FUNCTION_BLOCK "GCS7_E_MTRI"	// FB 57
TITLE = MTRI
//  
//COPYRIGHT:    (C) 1996 BY  BUHLER LTD.
//                           CH-9240 UZWIL  SWITZERLAND
//
//PRODUCT:      GCS7
//
//TITLE:        Element Control MTRI
//
//-------------------------------------------------------------------------
//
//IDENT:        AUTHOR:             DEPT:                       DATE:
//
//FB57.1.2      A.Egli              CT3                         18-Nov-2003
//              Handling Restdischarge
//FB57.1.1      A.Egli              CT3                         29-Sep-2003
//              Value in Units [1.00 to 8.00] = [-60° to 45°]
//FB57.1.0      A.Egli              CT3                         22-Apr-2003
//              1st Release in S7
//
//-------------------------------------------------------------------------
//
//PURPOSE:      MANUAL : see [MTRIxxMAN]
//
//RESTRICTIONS: S7
//
//-------------------------------------------------------------------------
//
//=======================================================
//Log Message: 
//------------------------------------------------------
//0   Stopped
//2   Adjusted
//9   fault cancelled
//10  emptied
//11  fault monitoring time
//12  fault adjusting time
//13  fault toloerance
//
//=======================================================
//StCode:  State               
//------------------------------------------------------
//32  StFault               
// 1  StStopped             
//41  StStopped.HWStop               StStopped + InHWStop
//51  StStopped.DPFault              StStopped + InDPFault
// 2  StAdjusting             
//12  StAdjusting.Calibration             
// 3  StAdjusted.Automatic              
//13  StAdjusted.Hand
//
AUTHOR : EA
FAMILY : GCS7LL
NAME : MTRI
VERSION : 1.2
VAR
  StCode : INT ;	//Element state code
  InEnable : BOOL ;	//Interlocking: 1=Enable to open /0=Intermediate closing
  CmdRestdischarge : BOOL ;	//Command to restdischarge
  CmdCalibration : BOOL ;	//Calibration 0 point
  InpMinus : BOOL ;	//Input button "Minus"
  InpPlus : BOOL ;	//Input button "Plus"
  CmdNewJob : BOOL ;	//Command new job
  InModeRemote : BOOL ;	//1=Target position from PC, 0=Target position with +/-
  spare27 : BOOL ;
  CmdOff : BOOL ;	//Pulse to stop  (manual mode)
  CmdOn : BOOL ;	//Pulse to start  (manual mode)
  CmdNext : BOOL ;	//Pulse to start element in automatic mode
  CmdFaultReset : BOOL ;	//Command to reset fault
  InLocal : BOOL ;	//1= Local mode (no fault by start with service switch)
  InManual : BOOL ;	//1= Manual/ 0= Automatic
  InReport : BOOL ;	//Report of all state transitions
  spare0207 : BOOL ;
  InHWStop : BOOL ;	//HW stop is detected, no fault
  InDPFault : BOOL ;	//DP-Fault is detected, no fault
  OutAutomatic : BOOL ;	//1=Automatic adjusting, 0=Position was change with +/-button
  OutRestdischargeDone : BOOL ;	//Restdischarge done
  OutpLampMinus : BOOL ;	//Lamp Minus
  OutpLampPlus : BOOL ;	//Lamp Plus
  OutpRunMinus : BOOL ;	//Motor in direction minus
  OutpRunPlus : BOOL ;	//Motor in direction plus
  StStopped : BOOL ;	//Element is stopped
  StAdjusting : BOOL ;	//Element is adjusting
  StAdjusted : BOOL ;	//Element is adjusted, motor is stopped
  StEmptying : BOOL ;	//Element is rotating 180° for restdischarge
  StFault : BOOL ;	//Element has a fault
  spare55 : BOOL ;
  spare56 : BOOL ;
  spare57 : BOOL ;
  OutRestdischargePosition : BOOL ;	//Resdischarge position was reached
  OutFinalAdjusting : BOOL ;	//Target positon was oversteped
  InpPosition : INT ;	//Input of sensor [Cray Code 10 Bit ]
  InPositionTargetUnit : INT ;	//In:    Target position [1.00  to  8.00 Unit]
  InOutPositionTargetDeg : INT ;	//In:    Target position [0.0 to +360.0 °]
  spare14 : INT ;
  OutPositionTargetDeg : INT ;	//Out: Target position [0.0 to +360.0 °]
  OutPositionActualUnit : INT ;	//Actual  position [1.00 to +8.00 Unit]
  OutPositionActualDeg : INT ;	//Actual  position [0.0 to +360.0 °]
  OutAlarmNrLog : INT ;	//Last textnumber send to log
  Par : STRUCT
   ParObjectNo : INT ;	//Is used for communication with PC, e.g. for message
   ParMsgType : INT ;	//Is used for message (translation of state)
   ParHornCode : INT ;	//Is used by horn module
   ParLogOff : BOOL ;	//Report is off
   ParManual : BOOL ;	//Manual mode without interlocking
   ParTolerance : INT  := 5;	//Tolerance position [0.1 Grad]
   ParMonTime : INT  := 20;	//Monitoring time until element change to StFault, if positon not changes
   ParAdjustingTime : INT  := 300;	//Monitoring time until element change to StFault , if not adjusted
   OutMonTime : INT ;	//Actual monitoring time
   OutAdjstingTime : INT ;	//Actual monitoring time
   CopyPositionTarget : INT ;	//Internal used
   CopyPositionActual : INT ;	//Internal used
  END_STRUCT ;
END_VAR
VAR_TEMP
  tmpLOGvalue : WORD ;	//LOG value
  tmpReport : BOOL ;	//Global LOG all
  tmpOpen : BOOL ;
  tmpOff : BOOL ;
  tmpLenDyn : DINT ;
  tmpMonFault : BOOL ;
  tmpAdjustingFault : BOOL ;
  tmpLocal : BOOL ;
  tmpLocalFault : BOOL ;
  tmpFault : BOOL ;
  tmpAdjusted : BOOL ;
  tmpLampMode1 : BOOL ;
  tmpLimitLow : INT ;
  tmpLimitHigh : INT ;
  tmpOutValue : INT ;
  tmpBitValue : INT ;
  tmpTarget : INT ;
  tmpValue : DINT ;
  tmpDelta : INT ;
  tmpForward : BOOL ;
  tmpAdjustedRecipe : BOOL ;	//Actual position is in tolerance of recipe position
  tmpNewTargetPos : BOOL ;	//Target position has changed
END_VAR
BEGIN
NETWORK
TITLE =  Start Global
      L     46;
      T     #tmpLenDyn;	//--> Len dynamic data in byte
NETWORK
TITLE = PC Control
//=== Test Object number =====================
      L     "SYS_DirectCtrlDB".PC.ObjectNo;	//PCControl.ObjectNo
      L     #Par.ParObjectNo;	//Input ObjectNo
      <>I;
      JC    Ctrl;
//=== Test OType      ========================
      L     1057;	//Input object type
      L     "SYS_DirectCtrlDB".PC.ObjectType;	//PCControl.ObjectType
      <>I;
      JC    Ctrl;
//=== Test Handshake =========================
      A     "SYS_DirectCtrlDB".PC.Hsk.FExamine;	// Handshake.FExamine
      JC    pExa;
      A     "SYS_DirectCtrlDB".PC.Hsk.FDefineCmd;	// Handshake.FDefineCmd
      JC    pCmd;
      A     "SYS_DirectCtrlDB".PC.Hsk.FDefinePara;	// Handshake.FDefinePara
      JC    pPar;
pIni: L     2;	// FcInit
      UC    "SYS_DirectCtrl";
      JU    Ctrl;
// Write parameter 
pPar: LAR1  P#DBX 58.0;	//PCControl.Value[1]
      L     P##Par;
      L     DW#16#FFFFF;
      AD;
      +AR1;
      L     DBW [AR1,P#8.0];
      T     #Par.ParTolerance;
      L     DBW [AR1,P#10.0];
      T     #Par.ParMonTime;
      L     DBW [AR1,P#12.0];
      T     #Par.ParAdjustingTime;
// Write new commands from PC to Interface of group 
pCmd: A     "SYS_DirectCtrlDB".PC.Cmd1[1];	//Cmd1[1]   =CmdRestdischarge
      S     #CmdRestdischarge;
      S     #CmdOn;
      A     "SYS_DirectCtrlDB".PC.Cmd1[2];	//Cmd1[2]   =CmdCalibration
      S     #CmdCalibration;
      A     "SYS_DirectCtrlDB".PC.Cmd1[5];	//Cmd1[5]   =CmdNewJob
      S     #CmdNewJob;
      A     "SYS_DirectCtrlDB".PC.Cmd1[6];	//Cmd1[6]   =CmdModeRemote
      S     #InModeRemote;
      A     "SYS_DirectCtrlDB".PC.Cmd2[6];	//Cmd2[6]   =CmdModeLocal
      R     #InModeRemote;
      A     "SYS_DirectCtrlDB".PC.Cmd1[8];	//Cmd1[8]   =CmdOff
      S     #CmdOff;
      A     "SYS_DirectCtrlDB".PC.Cmd1[9];	//Cmd1[9]   =CmdOn
      S     #CmdOn;
      A     "SYS_DirectCtrlDB".PC.Cmd1[10];	//Cmd1[10]   =CmdNext
      S     #CmdNext;
      A     "SYS_DirectCtrlDB".PC.Cmd1[11];	//Cmd1[11] =CmdFaultReset
      S     #CmdFaultReset;
      A     "SYS_DirectCtrlDB".PC.Cmd1[13];	//Cmd1[13] =CmdManualOn
      S     #InManual;
      A     "SYS_DirectCtrlDB".PC.Cmd2[13];	//Cmd2[13] =CmdManualOff
      R     #InManual;
      A     "SYS_DirectCtrlDB".PC.Cmd1[14];	//Cmd1[14]=CmdReportOn
      S     #InReport;
      A     "SYS_DirectCtrlDB".PC.Cmd2[14];	//Cmd2[14]=CmdReportOff
      R     #InReport;
      AN    "SYS_DirectCtrlDB".PC.Cmd1[9];	// CmdOn
      O     "GCS7_Gr_OutManualOff";	//Global.OutManualOff
      JC    pIni;
      L     0;
      L     "SYS_DirectCtrlDB".PC.Cmd3;	// "SYS_PCControl".PC.Cmd3
      ==I;
      JC    pIni;
      T     #InOutPositionTargetDeg;
      JU    pIni;
pExa: TAR2;	// Address Dynamic datas
      T     "SYS_DirectCtrlDB".GC.InDynAddr;	// -->PCControl.GC.InDynAddr
      L     #tmpLenDyn;	// Length Dynamic datas
      T     "SYS_DirectCtrlDB".GC.InDynLen;	// -->PCControl.GC.InDynLen
      L     0;
      T     "SYS_DirectCtrlDB".GC.InParaAddr;	// -->PCControl.GC.InParaAddr
      T     "SYS_DirectCtrlDB".GC.InParaLen;	// -->PCControl.GC.InParaLen
      L     1;	// Code FcExamine
      UC    "SYS_DirectCtrl";
      L     10;	//Revision
      T     "SYS_DirectCtrlDB".GC.Revision;
NETWORK
TITLE =  All State Init
//===Clear tmp Variable
//===Global Group Orders===
Ctrl: A     "GCS7_Gr_OutManualOn";	//Gr.OutManualOn
      S     #InManual;
      A     "GCS7_Gr_OutManualOff";	//Gr.OutManualOff
      R     #InManual;
      A     #InManual;
      S     "GCS7_Gr_InManual";	//Gr.InManualMode
//---Report is on---
      A     "GCS7_Gr_OutReportAll";	//Gr.OutReportAll
      O     #InReport;
      =     #tmpReport;
      A     #InLocal;
      AN    #InManual;
      =     #tmpLocalFault;
      A     #tmpLocalFault;
      O     #InHWStop;
      O     #InDPFault;
      =     #tmpLocal;
//---Enable---
      AN    #InEnable;
      AN    #InManual;
      O;
      AN    #InEnable;
      AN    #Par.ParManual;
      A     #InManual;
      O     #CmdOff;
      O     #tmpLocal;
      O     #StFault;
      =     #tmpOff;
//---Restdischarge---
      A     #OutRestdischargeDone;	//[1.2]
      R     #CmdRestdischarge;	//[1.2]
      A     #CmdNewJob;
      O     #CmdOn;
      O     #CmdOff;
      O     #tmpLocalFault;
      R     #OutRestdischargeDone;
      R     #OutRestdischargePosition;	//[1.2]
      R     #CmdRestdischarge;	//[1.2]
//---CmdCalibration---
      A     #CmdNewJob;
      O     #tmpLocalFault;
      O     #CmdOff;
      R     #CmdCalibration;
NETWORK
TITLE = Convert Actual position
      L     0;
      T     #tmpOutValue;
      L     1;
      T     #tmpBitValue;
      L     #InpPosition;	//GrayCode
      L     2#1111111111;
      AW;
      T     #tmpValue;
cLP1: L     0;
      L     #tmpValue;
      ==D;
      JC    cOUT;
      SRD   1;
      T     #tmpValue;
      JP    cIs1;	//Jump when Bit is 1
      JU    cNXT;
//Calculate, if bit is 1
cIs1: L     #tmpBitValue;
      SLD   1;
      L     #tmpOutValue;
      -D;
      L     1;
      -D;
      T     #tmpOutValue;
//======================
cNXT: L     #tmpBitValue;
      SLD   1;
      T     #tmpBitValue;
      JU    cLP1;
//Convert 0 to 1024 to 0 to +360.0
cOUT: L     #tmpOutValue;
      DTR;
      L     1.024000e+03;
      /R;
      L     3.600000e+03;
      *R;
      RND;
      T     #tmpOutValue;
      L     3600;
      L     #tmpOutValue;
      >=I;
      JC    cJ3;
      +     -3600;
cJ3:  T     #OutPositionActualDeg;
NETWORK
TITLE = Convert to Unit
// Convert target value
      L     #InPositionTargetUnit;
      ITD;
      L     500;	//Zero point =5.00
      -D;
      DTR;
      L     1.500000e+00;	//[0.1] Degree
      *R;
      RND;
      T     #InOutPositionTargetDeg;
      L     0;
      >=I;
      JC    cuJ0;
      TAK;
      L     3600;
      +I;
      T     #InOutPositionTargetDeg;
cuJ0: NOP   0;
// Convert actual value
      L     2850;
      L     #OutPositionActualDeg;
      >=I;
      JC    cuJ1;
      +     -3600;
cuJ1: ITD;
      DTR;
      L     1.500000e+00;	//[0.1] Degree
      /R;
      RND;
      +     500;	//Zero point =5.00
      T     #OutPositionActualUnit;
NETWORK
TITLE = Target position
      NOP   0;
//---OutRemote---
      L     #Par.CopyPositionTarget;
      L     #InOutPositionTargetDeg;
      T     #Par.CopyPositionTarget;
      T     #tmpTarget;
      <>I;
      O     #CmdNewJob;
      O     #CmdOn;
      S     #OutAutomatic;
      =     #tmpNewTargetPos;
      R     #OutFinalAdjusting;
//---Change to local Operation 
      A     #InpPlus;
      O     #InpMinus;
      ON    #InModeRemote;
      R     #OutAutomatic;
//---Target position
      L     #InOutPositionTargetDeg;
      A     #OutAutomatic;
      JC    TPJ1;
      A     #StEmptying;
      JC    TPEn;
      L     #OutPositionActualDeg;
TPJ1: T     #OutPositionTargetDeg;
TPEn: NOP   0;
NETWORK
TITLE = Check adjusted
      NOP   0;
//------------------------------
//Test adjusted
      L     #OutPositionActualDeg;
      L     #OutPositionTargetDeg;
      -I;
      JP    CAJ1;
      INVI;
CAJ1: T     #tmpValue;
      L     1800;
      <I;
      JC    CAJ2;
      L     3600;
      L     #tmpValue;
      -I;
      T     #tmpValue;
CAJ2: L     #tmpValue;
      L     #Par.ParTolerance;
      <=I;
      =     #tmpAdjusted;
//------------------------------
//Test adjusted in recipe position 
      L     #OutPositionTargetDeg;
      L     #InOutPositionTargetDeg;
      -I;
      JP    CBJ1;
      INVI;
CBJ1: T     #tmpValue;
      L     1800;
      <I;
      JC    CBJ2;
      L     3600;
      L     #tmpValue;
      -I;
      T     #tmpValue;
CBJ2: L     #tmpValue;
      L     #Par.ParTolerance;
      <=I;
      =     #tmpAdjustedRecipe;
NETWORK
TITLE = Monitoring time
      A     #OutpRunMinus;
      O     #OutpRunPlus;
      A(;
      L     #Par.CopyPositionActual;
      L     #OutPositionActualDeg;
      ==I;
      T     #Par.CopyPositionActual;
      );
      O     #OutFinalAdjusting;	//[1.1]
      JC    MTJ1;
      L     0;
      T     #Par.OutMonTime;
//---Count timer 
MTJ1: AN    #OutpRunMinus;
      AN    #OutpRunPlus;
      ON    "GCS7_Gr_OutTick200ms";	//Gr.OutTick200ms
      JC    MTJ2;
      L     #Par.OutMonTime;
      +     2;
      T     #Par.OutMonTime;
      L     #Par.OutAdjstingTime;
      +     2;
      T     #Par.OutAdjstingTime;
//---Monitoring Alarm 
MTJ2: L     #Par.ParMonTime;
      L     #Par.OutMonTime;
      <=I;
      AN    #CmdCalibration;
      AN    #tmpLocal;
      =     #tmpMonFault;	//Condition for fault
      L     #Par.ParAdjustingTime;
      L     #Par.OutAdjstingTime;
      <=I;
      A     #StAdjusting;
      AN    #tmpLocal;
      AN    #CmdCalibration;
      =     #tmpAdjustingFault;
      A     #tmpAdjustingFault;
      O     #tmpMonFault;	//Condition for fault
      =     #tmpFault;
NETWORK
TITLE = States
//===State machine===
      A     #StStopped;
      JC    S0;
      A     #StAdjusting;
      JC    S1;
      A     #StAdjusted;
      JC    S2;
      A     #StEmptying;
      JC    S3;
      A     #StFault;
      JC    S4;
      S     #StStopped;	// Init
      L     0;
      T     #Par.OutMonTime;
      JU    S0;
NETWORK
TITLE = StStopped
// Any transition to StClosed
xxS0: S     #StStopped;
      JU    LOG1;
//=== Logic ====
// Transition to StAdjusting
S0:   A     #CmdNext;
      AN    #InManual;
      O     #CmdOn;
      AN    #tmpOff;
      O     #CmdCalibration;
      O(;
      A     #InpMinus;
      O     #InpPlus;
      A     #tmpLocal;
      );
      R     #StStopped;
      JC    xxS1;
// Transition to fault
      A     #tmpFault;
      R     #StStopped;
      JC    xxS4;
      JU    OUT;
NETWORK
TITLE = StAdjusting
// Any transition to StOpening
xxS1: S     #StAdjusting;
      L     0;
      T     #Par.OutAdjstingTime;
      JU    OUT;
//=== Logic ====
// Transition for Stopped
S1:   A     #tmpOff;
      AN    #CmdCalibration;
      AN    #InpMinus;
      AN    #InpPlus;
      R     #StAdjusting;
      JC    xxS0;	//--> StStopped
// Transition for Emptying
      A     #CmdRestdischarge;
      AN    #CmdCalibration;
      R     #StAdjusting;
      JC    xxS3;	//--> StEmptying
// Transition for StAdjusted
      A     #tmpAdjusted;
      AN    #CmdCalibration;
      AN    #tmpLocal;
      AN    #InpPlus;
      AN    #InpMinus;
      R     #StAdjusting;
      JC    xxS2;	//--> StAdjusted
// Transition for StFault
      A     #tmpFault;
      R     #StAdjusting;
      L     B#(1, 11);	// Message ('Fault not open' )
      JC    xxS4;
      JU    OUT;
NETWORK
TITLE = StAdjusted
// Any transition to StCoarse
xxS2: S     #StAdjusted;
      JU    LOG1;
//=== Logic ====
// Transition to StAdjusting
S2:   AN    #tmpAdjusted;
      O     #InpPlus;
      O     #InpMinus;
      O     #CmdCalibration;
      R     #StAdjusted;
      JC    xxS1;	//--> StAdjusting
// Transition to StEmptying
      A     #CmdRestdischarge;
      AN    #tmpLocal;
      R     #StAdjusted;
      JC    xxS3;	//--> StEmptying
// Transition to StStopped
      A     #tmpOff;
      R     #StAdjusted;
      JC    xxS0;	//--> StStopped
// Transition for fault
      A     #tmpFault;
      R     #StAdjusted;
      JC    xxS4;
      JU    OUT;
NETWORK
TITLE = StEmptying
// Any Transition to StClosing
xxS3: S     #StEmptying;
      R     #OutRestdischargePosition;
      L     0;
      T     #Par.OutAdjstingTime;
      JU    OUT;
//=== Logic ====
S3:   L     #OutPositionTargetDeg;
      L     1820;
      -I;
      JP    S3J1;
      L     3600;
      +I;
S3J1: T     #tmpTarget;
//------------------------------
//Test adjusted
//------------------------------
      L     #OutPositionActualDeg;
      L     #tmpTarget;
      -I;
      JP    S3J2;
      INVI;
S3J2: T     #tmpDelta;
      L     1800;
      <I;
      JC    S3J3;
      L     3600;
      L     #tmpDelta;
      -I;
      T     #tmpDelta;
S3J3: L     #tmpDelta;
      L     10;	//1.0 grad
      <=I;
      S     #OutRestdischargePosition;
      L     #tmpTarget;
      AN    #OutRestdischargePosition;
      JC    S3J4;
      L     #OutPositionTargetDeg;
S3J4: T     #tmpTarget;
// Transition for StAdjusted
      A     #OutRestdischargePosition;
      A     #tmpAdjusted;
      S     #OutRestdischargeDone;
      R     #CmdRestdischarge;
      R     #StEmptying;
      S     #StAdjusted;
      JC    LOG1;
// Transition for StStopped         
      A     #tmpOff;
      O     #CmdNewJob;	//[1.2]
      R     #StEmptying;
      JC    xxS0;
// Transition for StFault
      A     #tmpFault;
      R     #StEmptying;
      JC    xxS4;
      JU    OUT;
NETWORK
TITLE = StFault
// Any transiton to Fault  
xxS4: S     "GCS7_Gr_InFaultFlag";	// Gr.InFaultFlag
      S     #StFault;
      CALL  "SYS_Horn_Code" (
           FcCode                   := 1,
           ParObjectType            := 1057,
           ParObjectNo              := #Par.ParObjectNo,
           ParHornCode              := #Par.ParHornCode);
      JU    LOGE;
//=== Logic ====
S4:   AN    #CmdFaultReset;
      AN    "GCS7_Gr_OutFaultReset";	// OutFaultReset
      AN    #tmpLocalFault;
      JC    OUT;
//Transition to StClosed
      R     #StFault;
      S     #StStopped;
      L     B#(3, 9);	// Message ('fault cancelled' )
      JU    LOG0;
NETWORK
TITLE = Log
LOG0: L     B#(3, 9);	// Message ('fault cancelled' )
      JU    LOG;
LOG1: AN    #tmpReport;
      JC    OUT;
      A     #StAdjusted;
      A     #OutRestdischargeDone;
      L     B#(1, 3);	// Message ('Emptied' )
      JC    LOG;
      A     #StAdjusted;
      L     B#(1, 2);	// Message ('Adjsuted' )
      JC    LOG;
      A     #StStopped;
      L     B#(1, 1);	// Message ('Stopped' )
      JC    LOG;
      JU    OUT;
//Transition to Fault
LOGE: A     #tmpMonFault;
      A     #OutFinalAdjusting;	//[1.1]
      L     B#(1, 13);	// Message ('Adjusting Tolerance' )
      JC    LOG;
      A     #tmpMonFault;
      L     B#(1, 11);	// Message ('Adjusting time' )
      JC    LOG;
      L     B#(1, 12);	// Message ('Timeout Adjusting Time' )
      JU    LOG;
LOG:  A     #Par.ParLogOff;	//---Set LOG Message
      JC    OUT;
      T     #tmpLOGvalue;
      L     W#16#FF;
      AW;
      T     #OutAlarmNrLog;
      CALL  "GCS7_LogConvert" (
           ObjectNo                 := #Par.ParObjectNo,
           MsgType                  := #Par.ParMsgType,
           ClassMsgTxt              := #tmpLOGvalue,
           OType                    := 1057);	// LOG Message Converter / Entry / Contains Class and TextNo
NETWORK
TITLE = Global End
OUT:  SET;	//---Clear all commands
      R     #CmdNewJob;
      R     #CmdOff;
      R     #CmdOn;
      R     #CmdNext;
      R     #CmdFaultReset;
//--Output for group 
      AN    #InLocal;
      O     #InManual;
      A     #InDPFault;
      S     "GCS7_Gr_InDPFault";
      AN    #InLocal;
      O     #InManual;
      A     #InHWStop;
      S     "GCS7_Gr_InHWStop";
NETWORK
TITLE = Output
      NOP   0;
      SET;
      S     #tmpForward;
//--Difference angle ----- 
      L     #tmpTarget;
      L     #OutPositionActualDeg;
      -I;
      JP    opJ1;	//--> Negativ
      NEGI;
      R     #tmpForward;
opJ1: T     #tmpValue;
      L     1800;
      <=D;
      JC    opJ2;
//IF angle is > 180 THEN Other way is shorter
      AN    #tmpForward;
      =     #tmpForward;
//--Change direction //[1.1] -->
opJ2: A     #tmpForward;
      A     #OutpRunMinus;
      O;
      AN    #tmpForward;
      A     #OutpRunPlus;
      S     #OutFinalAdjusting;
      A     #tmpNewTargetPos;
      ON    #OutAutomatic;
      ON    #StAdjusting;
      R     #OutFinalAdjusting;	// <---[1.1]
//-- OutRunPlus
      A     #tmpForward;
      AN    #tmpOff;
      A(;
      A     #StAdjusting;
      A     #OutAutomatic;
      O     #StEmptying;
      AN    #CmdCalibration;	//[1.1]
      );
      O(;
      A     #InpPlus;
      AN    #StEmptying;	//[1.1]
      );
      AN    #InpMinus;
      =     #OutpRunPlus;
//-- OutRunMinus
      AN    #tmpForward;
      AN    #tmpOff;
      A(;
      A     #StAdjusting;
      A     #OutAutomatic;
      O     #StEmptying;
      AN    #CmdCalibration;	//[1.1]
      );
      O(;
      A     #InpMinus;
      AN    #StEmptying;	//[1.1]
      );
      AN    #InpPlus;
      =     #OutpRunMinus;
NETWORK
TITLE = Lamps
      AN    #tmpAdjustedRecipe;
      ON    #InModeRemote;
      AN    #StStopped;
      AN    #tmpLocal;
      AN    #CmdCalibration;
      =     #tmpLampMode1;	//Lamps Flashing
      L     0;
      L     #OutPositionActualDeg;
      ==I;
      O(;
      L     1800;
      <I;
      A     "SYS_Pulse1000ms";
      );
      A     #CmdCalibration;	//0-Position Calibration ==> Lamp On
      O;
      A     #tmpLampMode1;
      A(;
      AN    #tmpAdjustedRecipe;
      A     #tmpForward;
      O     "SYS_Pulse1000ms";
      );
      =     #OutpLampMinus;
      L     0;
      L     #OutPositionActualDeg;
      ==I;
      O(;
      L     1800;
      >=I;
      A     "SYS_Pulse1000ms";
      );
      A     #CmdCalibration;	//0-Position Calibration ==> Lamp On
      O;
      A     #tmpLampMode1;
      A(;
      AN    #tmpForward;
      AN    #tmpAdjustedRecipe;
      ON    "SYS_Pulse1000ms";
      );
      =     #OutpLampPlus;
NETWORK
TITLE = State Code
      AN    #StStopped;
      JC    STC2;
      L     41;	//Code: StClosed.HWStop
      A     #InHWStop;
      JC    STC;
      L     51;	//Code: StClosed.DPFault
      A     #InDPFault;
      JC    STC;
      L     1;	// Code: closed
      JU    STC;
STC2: L     2;	// Code: StAdjusting
      A     #StAdjusting;
      AN    #CmdCalibration;
      JC    STC;
      L     12;	// Code: StAdjusting.Calibration
      A     #StAdjusting;
      A     #CmdCalibration;
      JC    STC;
      L     3;	// Code: StAdjusted.Remote
      A     #OutAutomatic;
      O     #tmpAdjustedRecipe;
      A     #StAdjusted;
      JC    STC;
      L     13;	// Code: StAdjusted.Local
      A     #StAdjusted;
      JC    STC;
      L     4;	// Code: StEmptying
      A     #StEmptying;
      JC    STC;
      L     32;	// Code: fault
STC:  L     #StCode;	// Old state code
      TAK;
      T     #StCode;	// Save state code
      <>I;
      L     3;	// Load code for CBit methode
      CC    "SYS_CBitCtrl";
END_FUNCTION_BLOCK

FUNCTION_BLOCK "GCS7_M_BCFA"	// FB 58
TITLE = Flaker
//COPYRIGHT:    (C) 2003  BUHLER AG, CH-9240 UZWIL, SWITZERLAND
//
//PRODUCT:      GCS7
//
//TITLE:        Machine Flaker Control 
//
//-------------------------------------------------------------------------
//
//IDENT:        AUTHOR:             DEPT:                       DATE:
//FB58.1.4      A.Smart             CDDP                        14-Apr-2004
//              It is possible now to give CmdReleaseEngage and
//              CmdSequenceStop at the same time to the BCFA, to trigger
//              the correct emptying out sequence.
//FB58.1.3      A.Smart             CDDP                        12-Aug-2003
//              New Signal InFeedRoll to release the feed roll of the flaker
//              There are particular situations where the flaker should stop
//              the feedroll. The plant control can only know this. 
//FB58.1.2      A.Smart             CDDP                        08-Jul-2003
//              New Signal InNewJobWait to decide whether to wait for the
//              Start Job Change Command from the BCFA machine
//              (it is not required when starting the line from completely empty)
//FB58.1.1      A.Smart             CDDP                        07-Jul-2003
//              Bug fix for Vibro Feeder and Flap Position
//FB58.1.0      A.Egli              CT3                         07-Apr-2003
//              1st Release
//-------------------------------------------------------------------------
//
//PURPOSE:      MANUAL : see [DICxxMAN]
//
//RESTRICTIONS: S7
//
//-------------------------------------------------------------------------
//=======================================================
//Log Message: 
//------------------------------------------------------
// 0  false
// 2  true
// 9  fault cancelled
//10  fault device
//11  fault true
//12  fault false
//13  prealarm true
//14  prealarm false
//
//=======================================================
//StCode:  State               
//------------------------------------------------------
//32  StFault                  StFault+InpFaultDev=0 
//31  StFault.DEV              StFault+InpFaultDev=1 
// 1  StFalse               
//11  StFalse.Warning          StFalse+OutWarning
//41  StFalse.HWStop           StFalse+HWStop 
//51  StFalse.DPFault          StFalse+DPFault
//61  StFalse.FaultDev         InLocal=1 +InpFaultDef +InpTrue=0
// 2  StCtoTrue             
//12  StCtoTrue.Warning     
// 3  StTrue                
//13  StTrue.Warning           StTrue+OutWarning
//43  StTrue.HWStop            StTrue+InHWStop
//53  StTrue.DPFault           StTrue+InDPFault
//63  StTrue.FaultDev          InLocal=1 +InpFaultDef +InpTrue=1
// 4  StCtoFalse             
//14  StCtoFalse.Warning       StCtoFalse+OutWarning
//
//
//
AUTHOR : EA
FAMILY : GCS7LL
NAME : BCFA
VERSION : 1.4
VAR
  Ma : STRUCT
   StCode : INT ;	//Element state code
   InEnable : BOOL ;	//Enable to run the element reverse
   InEngage : BOOL ;	//Enable to run engage
   InNewJobWait : BOOL ;	//Signal to wait for Start Job Change from the Operator
   InFeedRoll : BOOL ;	//Enable to run the feed roll of the flaker
   spare24 : BOOL ;
   CmdNewJob : BOOL ;	//Pulse to start the element in automatic mode (see global flags)
   spare26 : BOOL ;
   spare27 : BOOL ;
   CmdOff : BOOL ;	//Pulse to stop the element immediately (manual mode)
   CmdOn : BOOL ;	//Pulse to start the element immediately (manual mode)
   CmdNext : BOOL ;	//Pulse to start the element in automatic mode (see global flags)
   CmdFaultReset : BOOL ;	//Command to reset fault
   InLocal : BOOL ;	//1= Local mode (no fault by start with service switch)
   InManual : BOOL ;	//1= Manual/ 0=Automatic
   InReport : BOOL ;	//Report of all state transitions
   InSeqStop : BOOL ;	//Stop automatically after idling time
   spare40 : BOOL ;
   spare41 : BOOL ;
   InSimulation : BOOL ;	//DP:
   OutComFault : BOOL ;	//Communication fault
   spare44 : BOOL ;
   spare45 : BOOL ;
   spare46 : BOOL ;
   OutWarning : BOOL ;	//Warning
   StStopped : BOOL ;	//BCFA in state Automatic.Stopped
   StStarting : BOOL ;	//BCFA in state Automatic.Starting
   StProduction : BOOL ;	//BCFA in state Automatic.Production
   StStopping : BOOL ;	//BCFA in state Automatic.Stopping
   StFaultCom : BOOL ;
   StStandby : BOOL ;	//BCFA in state Automatic.Standby
   StService : BOOL ;	//BCFA is in mode Servive or Neutral
   OutFaulted : BOOL ;	//Fault
   ToBCFA : STRUCT
    SP_GapLeft : INT ;	//Setpoint gap left
    SP_GapRight : INT ;	//Setpoint gap right
    SP_TempRoll : INT ;	//Setpoint water temperture
    SP_FE_RollSpeed : INT ;	//Setpoint speed roll feeder
    SP_FE_VibroSpeed : INT ;	//Setpoint speed vibro feeder
    SP_RC_Option : INT ;	//Setpoint roll cooling option (1 = with, 2 = without)
    res120 : INT ;
    res140 : INT ;
    res160 : INT ;
    res180 : INT ;
    CmdSequenceStart : BOOL ;	//Start flaker
    CmdSequenceStop : BOOL ;	//Sequence stop flaker
    CmdReleaseEngage : BOOL ;	//Plant release signal for engaging (=> E0.0) (e.q. release roll engage on site)
    CmdDoneJobchange : BOOL ;	//Job change executed
    CmdReleaseFeed : BOOL ;	//Plant release signal for feed roll
    res205 : BOOL ;
    res206 : BOOL ;
    res207 : BOOL ;
    res210 : BOOL ;
    res211 : BOOL ;
    res212 : BOOL ;
    res213 : BOOL ;
    res214 : BOOL ;
    res215 : BOOL ;
    res216 : BOOL ;
    res217 : BOOL ;
    res220 : WORD ;
    res240 : WORD ;
    res260 : WORD ;
    res280 : WORD ;
    LineCheck : WORD ;	//Line check value from remote
   END_STRUCT ;
   FromBCFA1 : STRUCT
    RV_GapLeft : INT ;	//Actual gap value left
    RV_GapRight : INT ;	//Actual gap value right
    RV_TempRoll : INT ;	//Actual water temperature
    RV_MM_1_Current : INT ;	//Actual current mainmotor 1
    RV_MM_2_Current : INT ;	//Actual current mainmotor 2
    RV_ForceLeft : INT ;	//Actual roll force left
    RV_ForceRight : INT ;	//Actual roll force right
    RV_FE_DSDC_Temp : INT ;	//Actual conditioner temperature
    res480 : INT ;
    RV_SP_GapLeft : INT ;	//Actual setpoint gap left
    RV_SP_GapRight : INT ;	//Actual setpoint gap right
    RV_SP_TempRoll : INT ;	//Actual setpoint water temperture
    RV_SP_FE_RollSpeed : INT ;	//Actual setpoint speed roll feeder
    RV_SP_FE_VibroSpeed : INT ;	//Actual setpoint speed vibro feeder
    RV_SP_RC_Option : INT ;	//Actual setpoint roll cooling option (1 = with, 2 = without)
    res620 : INT ;
   END_STRUCT ;
   FromBCFA2 : STRUCT
    Sta_Automatic : BYTE ;	//Status automatic mode
    Sta_Calibration : BYTE ;	//Status calibration mode
    Sta_OperationMode : BYTE ;	//Status operation mode
    Sta_MM_1_On : BOOL ;	//Mainmotor 1 running
    Sta_MM_1_Fault : BOOL ;	//Mainmotor 1 fault
    Sta_MM_2_On : BOOL ;	//Mainmotor 2 running
    Sta_MM_2_Fault : BOOL ;	//Mainmotor 2 fault
    Sta_ROLL_On : BOOL ;	//Roll feeder running
    Sta_ROLL_Fault : BOOL ;	//Roll feeder fault
    Sta_Vibro_On : BOOL ;	//Vibro channel running
    Sta_Vibro_Fault : BOOL ;	//Vibro cahnnel fault
    Sta_RC_On : BOOL ;	//Roll cooling on
    Sta_RC_Fault : BOOL ;	//Roll cooling fault
    Sta_HD_On : BOOL ;	//Hydraulic running
    Sta_HD_Fault : BOOL ;	//Hydraulic fault
    Sta_Engaged_On : BOOL ;	//Roll position engaged
    Sta_Engaged_Fault : BOOL ;	//Roll position fault
    Sta_Flap_Production : BOOL ;	//Outlet flap production (DSDC option)
    Sta_Flap_Fault : BOOL ;	//Outlet flap fault (DSDC option)
    Sta_Flow_Ok : BOOL ;	//Flow detector ok
    Sta_Flow_Fault : BOOL ;	//Flow detector fault
    res700 : WORD ;
    res702 : WORD ;
    CmdStartJobchange : BOOL ;	//Start job change
    res741 : BOOL ;
    res742 : BOOL ;
    res743 : BOOL ;
    res744 : BOOL ;
    res745 : BOOL ;
    res746 : BOOL ;
    res747 : BOOL ;
    res750 : BYTE ;
    Alarm : STRUCT 	//Aux. signal to retry fault message
     A01System : BOOL ;
     A02Memory : BOOL ;
     A03SerialCom : BOOL ;
     A04MainMotor : BOOL ;
     A05MMotor1Range : BOOL ;
     A06MMotor2Range : BOOL ;
     A07Hydraulic : BOOL ;
     A08HydrPressTOut : BOOL ;
     A09 : BOOL ;
     A10GapAdjMotor : BOOL ;
     A11GapLeftEdpos : BOOL ;
     A12GapLeftRange : BOOL ;
     A13GapRightEndpos : BOOL ;
     A14GapRightRange : BOOL ;
     A15 : BOOL ;
     A16DryRunning : BOOL ;
     A17ProductNokWA : BOOL ;
     A18ProductNokAL : BOOL ;
     A19FeederMotor : BOOL ;
     A20WaterFlow : BOOL ;
     A21RollTpWA : BOOL ;
     A22RollTpMax : BOOL ;
     A23WaterTpRange : BOOL ;
     A24CondTpMinWA : BOOL ;
     A25CondTpMinAL : BOOL ;
     A26AirPressure : BOOL ;
     A27CondTpRange : BOOL ;
     A28ForceLeftRange : BOOL ;
     A29ForceRightRange : BOOL ;
     A30 : BOOL ;
     A31ProtectionKnife : BOOL ;
     A32ProtectionCover : BOOL ;
    END_STRUCT ;
    Message : DWORD ;
    res840 : WORD ;
    res860 : WORD ;
    res880 : WORD ;
    res900 : WORD ;
    res920 : WORD ;
    LineCheck : WORD ;	//Line check value to remote
   END_STRUCT ;
   OutAlarmNr : INT ;	//Is read from MEAF ; Is transformed for MWEB like MEAF
   OutAlarmNrLog : INT ;	//Last textnumber send to log
   Par : STRUCT
    ParObjectNo : INT ;	//Is used for communication with PC, e.g. for message
    ParMsgType : INT ;	//Is used for message (translation of state)
    ParHornCode : INT ;	//Is used by horn module
    ParLogOff : BOOL ;	//Report is off
    ParManual : BOOL ;	//Manual mode without interlocking
    ParIOByteNr : INT ;	//Address of first input and output byte
    ParSpare : INT ;
    CopyData : STRUCT
     Alarm : DWORD ;
     SP_GapLeft : INT ;	//Setpoint gap left
     SP_GapRight : INT ;	//Setpoint gap right
     SP_TempRoll : INT ;	//Setpoint water temperture
     SP_FE_RollSpeed : INT ;	//Setpoint speed roll feeder
     SP_FE_VibroSpeed : INT ;	//Setpoint speed vibro feeder
     SP_RC_Option : INT ;	//Setpoint roll cooling option (1 = with, 2 = without)
     res120 : INT ;
     res140 : INT ;
    END_STRUCT ;
    OutHelpFlags : STRUCT 	//Aux. signal to retry fault message
     OutComFaultRead : BOOL ;
     OutComFaultSend : BOOL ;
     OutFaultedMsg : BOOL ;
     OutComFaultMsg : BOOL ;
    END_STRUCT ;
   END_STRUCT ;
  END_STRUCT ;
  Motor1 : FB 12;
  Motor2 : FB 12;
  Hydraulic : FB 12;
  Cooler : FB 12;
  Engaged : FB 12;
  RollFeeder : FB 12;
  VibroFeeder : FB 12;
  Flap : FB 13;
  ProductFlow : FB 14;
END_VAR
VAR_TEMP
  Src : ANY ;	//Must by at LB0
  tmpSendData : STRUCT
   SP_GAP_LEFT : INT ;	//Setpoint gap left
   SP_GAP_RIGHT : INT ;	//Setpoint gap right
   SP_TEMP_ROLL : INT ;	//Setpoint water temperture
   SP_FE_ROLL_SPEED : INT ;	//Setpoint speed roll feeder
   SP_FE_VIBRO_SPEED : INT ;	//Setpoint speed vibro feeder
   SP_RC_OPTION : INT ;	//Setpoint roll cooling option (1 = with, 2 = without)
   res120 : INT ;
   res140 : INT ;
   res160 : INT ;
   res180 : INT ;
   CMD_SEQUENCE_START : BOOL ;	//Start flaker
   CMD_SEQUENCE_STOP : BOOL ;	//Sequence stop flaker
   CMD_RELEASE : BOOL ;	//Plant release signal (=> E0.0) (e.q. release roll engage on site)
   CMD_DONE_JOBCHANGE : BOOL ;	//Job change executed
   res204 : BOOL ;
   res205 : BOOL ;
   res206 : BOOL ;
   res207 : BOOL ;
   res210 : BOOL ;
   res211 : BOOL ;
   res212 : BOOL ;
   res213 : BOOL ;
   res214 : BOOL ;
   res215 : BOOL ;
   res216 : BOOL ;
   res217 : BOOL ;
   res220 : WORD ;
   res240 : WORD ;
   res260 : WORD ;
   res280 : WORD ;
   GET_LINE_CHECK : WORD ;	//Line check value from remote
  END_STRUCT ;
  tmpLOGvalue : WORD ;	//LOG value
  tmpAddr1 : WORD ;	//Number of the actual FB
  tmpAddr2 : WORD ;	//Number of the actual FB
  tmpReport : BOOL ;	//Global LOG all
  tmpFault : BOOL ;
  tmpLocal : BOOL ;
  tmpReturn1 : INT ;
  tmpReturn2 : INT ;
  tmpLenDyn : INT ;
  tmpValue : DINT ;
  error : INT ;
  tmpAddrAlarm : DINT ;
  tmpAddrCopyAlarm : DINT ;
  tmpAlarmNr : INT ;
  tmpCopyAlarm : DWORD ;
  tmpALARM : STRUCT 	//Aux. signal to retry fault message
   A01System : BOOL ;
   A02Memory : BOOL ;
   A03SerialCom : BOOL ;
   A04MainMotor : BOOL ;
   A05MMotor1Range : BOOL ;
   A06MMotor2Range : BOOL ;
   A07Hydraulic : BOOL ;
   A08HydrPressTOut : BOOL ;
   A09 : BOOL ;
   A10GapAdjMotor : BOOL ;
   A11GapLeftEdpos : BOOL ;
   A12GapLeftRange : BOOL ;
   A13GapRightEndpos : BOOL ;
   A14GapRightRange : BOOL ;
   A15 : BOOL ;
   A16DryRunning : BOOL ;
   A17ProductNokWA : BOOL ;
   A18ProductNokAL : BOOL ;
   A19FeederMotor : BOOL ;
   A20WaterFlow : BOOL ;
   A21RollTpWA : BOOL ;
   A22RollTpMax : BOOL ;
   A23WaterTpRange : BOOL ;
   A24CondTpMinWA : BOOL ;
   A25CondTpMinAL : BOOL ;
   A26AirPressure : BOOL ;
   A27CondTpRange : BOOL ;
   A28ForceLeftRange : BOOL ;
   A29ForceRightRange : BOOL ;
   A30 : BOOL ;
   A31ProtectionKnife : BOOL ;
   A32ProtectionCover : BOOL ;
  END_STRUCT ;
  tmpEnable : BOOL ;
END_VAR
BEGIN
NETWORK
TITLE =  Start Global
      L     110;
      T     #tmpLenDyn;
//Pointer  P##FromBCFA2.ALARM
      TAR2;
      L     P#82.0;	//  P##FromBCFA2.ALARM 
      +D;
      T     #tmpAddrAlarm;
//Pointer  P##tmpAddrCopyAlarm
      L     P##tmpCopyAlarm;
      T     #tmpAddrCopyAlarm;
//Copy Old Alarm Pattern
      L     #Ma.Par.CopyData.Alarm;
      T     #tmpCopyAlarm;
NETWORK
TITLE = PC Control
//=== Test Object number =====================
      L     "SYS_DirectCtrlDB".PC.ObjectNo;	//PCControl.ObjectNo
      L     #Ma.Par.ParObjectNo;	//Input ObjectNo
      <>I;
      JC    CTRL;
//=== Test OType      ========================
      L     2058;	//Input object type
      L     "SYS_DirectCtrlDB".PC.ObjectType;	//PCControl.ObjectType
      <>I;
      JC    CTRL;
//=== Test Handshake =========================
      A     "SYS_DirectCtrlDB".PC.Hsk.FExamine;	//Handshake.FExamine
      JC    pExa;
      A     "SYS_DirectCtrlDB".PC.Hsk.FDefineCmd;	//Handshake.FDefineCmd
      JC    pCmd;
      A     "SYS_DirectCtrlDB".PC.Hsk.FDefinePara;	//Handshake.FDefinePara
      JC    pPar;
      JC    CTRL;	//[1.1]
pIni: L     2;	//FcInit
      UC    "SYS_DirectCtrl";
      JU    CTRL;
//Write parameter 
pPar: NOP   0;
//Write new commands from PC to Interface of group 
pCmd: A     "SYS_DirectCtrlDB".PC.Cmd1[5];	//Cmd1[5]  =CmdNewJob
      S     #Ma.CmdNewJob;
      A     "SYS_DirectCtrlDB".PC.Cmd1[1];	//Cmd1[1]  =CmdEngage
      S     #Ma.InEngage;
      A     "SYS_DirectCtrlDB".PC.Cmd2[1];	//Cmd1[1]  =CmdDisengage
      R     #Ma.InEngage;
      A     "SYS_DirectCtrlDB".PC.Cmd1[8];	//Cmd1[8]  =CmdOff
      S     #Ma.CmdOff;
      A     "SYS_DirectCtrlDB".PC.Cmd1[9];	//Cmd1[9]  =CmdOn
      S     #Ma.CmdOn;
      A     "SYS_DirectCtrlDB".PC.Cmd1[11];	//Cmd1[11] =CmdFaultReset
      S     #Ma.CmdFaultReset;
      A     "SYS_DirectCtrlDB".PC.Cmd1[13];	//Cmd1[13] =CmdManualOn
      S     #Ma.InManual;
      A     "SYS_DirectCtrlDB".PC.Cmd2[13];	//Cmd2[13] =CmdManualOff
      R     #Ma.InManual;
      A     "SYS_DirectCtrlDB".PC.Cmd1[14];	//Cmd1[14] =CmdReportOn
      S     #Ma.InReport;
      A     "SYS_DirectCtrlDB".PC.Cmd2[14];	//Cmd2[14] =CmdReportOff
      R     #Ma.InReport;
      JU    pIni;
pExa: TAR2;	//Address dynamic datas
      T     "SYS_DirectCtrlDB".GC.InDynAddr;	//-->PCControl.GC.InDynAddr
      L     #tmpLenDyn;	//Length dynamic datas
      T     "SYS_DirectCtrlDB".GC.InDynLen;	//-->PCControl.GC.InDynLen
      L     0;
      T     "SYS_DirectCtrlDB".GC.InParaAddr;	//-->PCControl.GC.InParaAddr
      T     "SYS_DirectCtrlDB".GC.InParaLen;	//-->PCControl.GC.InParaLen
      L     1;	//Code FcExamine
      UC    "SYS_DirectCtrl";
      L     10;	//Revision
      T     "SYS_DirectCtrlDB".GC.Revision;
CTRL: NOP   0;
NETWORK
TITLE = (Profibus) Read data and store Data 
      L     #Ma.Par.ParIOByteNr;
      T     #tmpAddr1;
      +     32;
      T     #tmpAddr2;
      A     #Ma.InSimulation;
      JC    rSim;
      CALL  "SIEMENS_DPRD_DAT" (
           LADDR                    := #tmpAddr1,
           RET_VAL                  := #tmpReturn1,
           RECORD                   := #Ma.FromBCFA1);
      CALL  "SIEMENS_DPRD_DAT" (
           LADDR                    := #tmpAddr2,
           RET_VAL                  := #tmpReturn2,
           RECORD                   := #Ma.FromBCFA2);
      L     #tmpReturn1;
      L     0;
      <>I;
      O(;
      L     #tmpReturn2;
      L     0;
      <>I;
      );
      =     #Ma.Par.OutHelpFlags.OutComFaultRead;
      JU    rcv0;
//read from Simulation
rSim: R     #Ma.Par.OutHelpFlags.OutComFaultRead;
      A     "GCS7_Gr_SimDPtoImage";
      L     P#I 0.0;
      JC    rDB1;
      OPN   "TEST_IOSimuliInput";
      L     P#DBX 0.0;
rDB1: L     #Ma.Par.ParIOByteNr;
      SLD   3;
      +D;
      T     LD 6;	//->Src.BitAddress 
      L     W#16#1002;	//S7 word
      T     LW 0;	//->Src.type
      L     32;	//Length in byte
      T     LW 2;	//->Src.factor
      L     DBNO;
      A     "GCS7_Gr_SimDPtoImage";
      JC    rDB2;
      L     0;
rDB2: T     LW 4;	//->Src.DB
      CALL  "SIEMENS_BLKMOV" (
           SRCBLK                   := #Src,
           RET_VAL                  := #error,
           DSTBLK                   := #Ma.FromBCFA1);
      L     LD 6;	//->Src.BitAddress 
      L     P#32.0;
      +D;
      T     LD 6;	//->Src.BitAddress 
      CALL  "SIEMENS_BLKMOV" (
           SRCBLK                   := #Src,
           RET_VAL                  := #error,
           DSTBLK                   := #Ma.FromBCFA2);
rcv0: NOP   0;
NETWORK
TITLE =  All State Init
      NOP   0;
//===Global Group Orders===
      A     "GCS7_Gr_OutManualOn";	//Gr.OutManualOn
      S     #Ma.InManual;
      A     "GCS7_Gr_OutManualOff";	//Gr.OutManualOff
      R     #Ma.InManual;
      A     #Ma.InManual;
      S     "GCS7_Gr_InManual";	//Gr.InManualMode
//---FaultReset is on---
      A     "GCS7_Gr_OutFaultReset";	//Gr.OutOutFaultReset
      S     #Ma.CmdFaultReset;
//---Report is on---
      A     "GCS7_Gr_OutReportAll";	//Gr.OutReportAll
      O     #Ma.InReport;
      =     #tmpReport;
//---Local---
      A     #Ma.InLocal;
      AN    #Ma.InManual;
      =     #tmpLocal;
//---tmpEnable---
      A     #Ma.InEnable;
      O     #Ma.Par.ParManual;
      AN    #Ma.CmdOff;
      A     #Ma.InManual;
      O;
      AN    #Ma.InManual;
      A     #Ma.InEnable;
      =     #tmpEnable;
//--- New Job
      A     #Ma.CmdNewJob;	// 1.2
      A(;	// 1.2
      A     #Ma.FromBCFA2.CmdStartJobchange;	// 1.2
      ON    #Ma.InNewJobWait;	// 1.2
      );	// 1.2
      JCN   iEnd;	// 1.2
      SET;	// 1.2
      R     #Ma.CmdNewJob;
      L     0;
      T     #Ma.Par.CopyData.SP_GapLeft;
      T     #Ma.Par.CopyData.SP_GapRight;
      T     #Ma.Par.CopyData.SP_TempRoll;
      T     #Ma.Par.CopyData.SP_FE_RollSpeed;
      T     #Ma.Par.CopyData.SP_FE_VibroSpeed;
      T     #Ma.Par.CopyData.SP_RC_Option;
iEnd: NOP   0;
NETWORK
TITLE = Status to ASW
      NOP   0;
//=======================================
//OutComFault 
//=======================================
      A     #Ma.Par.OutHelpFlags.OutComFaultRead;
      O     #Ma.Par.OutHelpFlags.OutComFaultSend;
      O     #Ma.OutComFault;
      AN    #tmpLocal;
      AN    #Ma.CmdFaultReset;
      =     #Ma.OutComFault;
//=======================================
//Fault   
//=======================================
// --- Copy FromBCFA2.ALARM to tmpAlarm
      L     DID [#tmpAddrAlarm];	//FromBCFA2.ALARM
      LAR1  P##tmpALARM;
      T     LD [AR1,P#0.0];	//-->tmpAlarm
// --- Reset Warning bits in tmpAlarm
      SET;
      R     #tmpALARM.A17ProductNokWA;
      R     #tmpALARM.A21RollTpWA;
      R     #tmpALARM.A24CondTpMinWA;
// --- Check Faulted
      LAR1  P##tmpALARM;
      L     LD [AR1,P#0.0];	//tmpAlarm
      L     0;
      <>D;
      A(;
      L     #Ma.FromBCFA2.Sta_Automatic;
      L     1;	//Stopped
      ==I;
      O(;
      L     #Ma.FromBCFA2.Sta_Automatic;
      L     5;	//Stopping
      ==I;
      );
      );
      O     #Ma.OutComFault;
      AN    #tmpLocal;
      =     #Ma.OutFaulted;
// --- Check Warning
      L     DID [#tmpAddrAlarm];	//FromBCFA2.ALARM
      L     0;
      <>D;
      AN    #Ma.OutFaulted;
      AN    #tmpLocal;
      =     #Ma.OutWarning;
//=======================================
//Command for BCFA
//=======================================
      A     #Ma.CmdNext;
      AN    #Ma.InManual;
      O     #Ma.CmdOn;
      O     #Ma.ToBCFA.CmdSequenceStart;
      A     #tmpEnable;
      =     #Ma.ToBCFA.CmdSequenceStart;
      A     #Ma.InSeqStop;
      AN    #Ma.InManual;
      =     #Ma.ToBCFA.CmdSequenceStop;
      A     #Ma.CmdNext;
      AN    #Ma.InSeqStop;	// [1.4]
      AN    #Ma.InManual;
      O     #Ma.CmdOn;
      O     #Ma.ToBCFA.CmdReleaseEngage;
      A     #tmpEnable;
      A     #Ma.InEngage;
//      AN    #Ma.InSeqStop             // [1.4]
      =     #Ma.ToBCFA.CmdReleaseEngage;
      A     #Ma.FromBCFA2.CmdStartJobchange;
      =     #Ma.ToBCFA.CmdDoneJobchange;
      A     #Ma.InFeedRoll;	// [1.3]
      =     #Ma.ToBCFA.CmdReleaseFeed;	// [1.3]
NETWORK
TITLE =  StFault
      A     #Ma.OutComFault;
      =     #Ma.StFaultCom;
NETWORK
TITLE =  StService
      L     #Ma.FromBCFA2.Sta_OperationMode;
      L     1;	//Neutral
      ==I;
      O(;
      L     #Ma.FromBCFA2.Sta_OperationMode;
      L     2;	//Service
      ==I;
      );
      AN    #Ma.StFaultCom;
      FP    #Ma.StService;
      JC    LOGX;
NETWORK
TITLE =  StStopped
      L     #Ma.FromBCFA2.Sta_Automatic;
      L     1;
      ==I;
      AN    #Ma.StFaultCom;
      AN    #Ma.StService;
      FP    #Ma.StStopped;
      R     #Ma.ToBCFA.CmdSequenceStart;
      R     #Ma.ToBCFA.CmdReleaseEngage;
      JC    LOGX;
NETWORK
TITLE =  StStarting
      L     #Ma.FromBCFA2.Sta_Automatic;
      L     2;
      ==I;
      AN    #Ma.StFaultCom;
      AN    #Ma.StService;
      =     #Ma.StStarting;
NETWORK
TITLE =  StStandby
      L     #Ma.FromBCFA2.Sta_Automatic;
      L     3;
      ==I;
      AN    #Ma.StFaultCom;
      AN    #Ma.StService;
      =     #Ma.StStandby;
NETWORK
TITLE =  StProduction
      L     #Ma.FromBCFA2.Sta_Automatic;
      L     4;
      ==I;
      AN    #Ma.StFaultCom;
      AN    #Ma.StService;
      FP    #Ma.StProduction;
      JC    LOGX;
NETWORK
TITLE =  StStopping
      L     #Ma.FromBCFA2.Sta_Automatic;
      L     5;
      ==I;
      AN    #Ma.StFaultCom;
      AN    #Ma.StService;
      =     #Ma.StStopping;
NETWORK
TITLE = LOG
      NOP   0;
//-- Transition to Faulted
      A     #Ma.OutFaulted;
      AN    #Ma.Par.OutHelpFlags.OutFaultedMsg;
      JCN   S4;
//--Transition to StFault----
      S     #Ma.Par.OutHelpFlags.OutFaultedMsg;
      S     "GCS7_Gr_InFaultFlag";	//Gr.InFaultFlag
      CALL  "SYS_Horn_Code" (
           FcCode                   := 1,
           ParObjectType            := 2058,
           ParObjectNo              := #Ma.Par.ParObjectNo,
           ParHornCode              := #Ma.Par.ParHornCode);
//---Condition for Fault Cancelled
S4:   A     #Ma.OutFaulted;
      FN    #Ma.Par.OutHelpFlags.OutFaultedMsg;
      L     B#(4, 0);	//Message ('fault cancelled')
      JC    LOG;
//--------------------
//Log Alarm Communication
//--------------------
      L     B#(1, 96);
      A     #Ma.OutComFault;
      AN    #tmpLocal;
      FP    #Ma.Par.OutHelpFlags.OutComFaultMsg;
      JC    LOG;
//--------------------
//LOG Alarm message
//--------------------
      L     #tmpCopyAlarm;
      L     DID [#tmpAddrAlarm];	//FromBCFA2.ALARM
      AD;
      T     #tmpCopyAlarm;	//CopyData.ALARM
      L     0;
      L     DID [#tmpAddrAlarm];	//FromBCFA2.ALARM
      ==D;
      O     #tmpLocal;
      JC    M014;
      L     #tmpCopyAlarm;	//CopyData.ALARM
      ==D;
      JC    M014;	//-->No new Alarm
      L     1;
      T     #tmpAlarmNr;
M032: A     DIX [#tmpAddrAlarm];	//FromBCFA2.ALARM
      AN    L [#tmpAddrCopyAlarm];	//CopyData.ALARM
      S     L [#tmpAddrCopyAlarm];	//CopyData.ALARM
      JC    M033;
      L     #tmpAddrAlarm;
      +     L#1;
      T     #tmpAddrAlarm;
      L     #tmpAddrCopyAlarm;
      +     L#1;
      T     #tmpAddrCopyAlarm;
      L     #tmpAlarmNr;
      +     1;
      T     #tmpAlarmNr;
      L     32;
      <=I;
      JC    M032;	//-->Loop Alarm
      JU    M014;	//-->No new Alarm
//Alarm-Nr 1..80
M033: L     #tmpAlarmNr;
      T     #Ma.OutAlarmNr;
      L     B#(1, 0);
      OW;
      JU    LOG;	//Alarms 1..80
//===============================================
//State Transition
LOGX: AN    #tmpReport;
      JC    M014;
      A     #Ma.StStopped;
      L     B#(4, 91);	//Message ('Stopped')
      JC    LOG;
      A     #Ma.StProduction;
      L     B#(4, 94);	//Message ('Production')
      JC    LOG;
      A     #Ma.StService;
      L     B#(4, 95);	//Message ('Service')
      JC    LOG;
      JC    M014;
LOG:  A     #Ma.Par.ParLogOff;	//---Set LOG Message
      JC    M014;
      T     #tmpLOGvalue;
      L     W#16#FF;
      AW;
      T     #Ma.OutAlarmNrLog;
      CALL  "GCS7_LogConvert" (
           ObjectNo                 := #Ma.Par.ParObjectNo,
           MsgType                  := #Ma.Par.ParMsgType,
           ClassMsgTxt              := #tmpLOGvalue,
           OType                    := 2058);	//LOG Message Converter / Entry / Contains Class and TextNo
NETWORK
TITLE = Global End
//---Clear commands
M014: SET;
      R     #Ma.CmdFaultReset;
      R     #Ma.CmdNext;
      R     #Ma.CmdOn;
      R     #Ma.CmdOff;
      L     #tmpCopyAlarm;
      T     #Ma.Par.CopyData.Alarm;
NETWORK
TITLE = (Profibus) Send Data
      NOP   0;
//---------------------------
//Prepare Send Data
//---------------------------
      L     #Ma.FromBCFA2.LineCheck;
      T     #Ma.ToBCFA.LineCheck;
      CALL  "SIEMENS_BLKMOV" (
           SRCBLK                   := #Ma.ToBCFA,
           RET_VAL                  := #tmpReturn1,
           DSTBLK                   := #tmpSendData);
//---------------------------
//Send only value with modification
//---------------------------
// --Value1
      L     #Ma.Par.CopyData.SP_GapLeft;
      L     #Ma.ToBCFA.SP_GapLeft;
      <>I;
      AN    #Ma.CmdNewJob;
      JC    M018;
      L     0;
M018: T     #tmpSendData.SP_GAP_LEFT;
      L     #Ma.ToBCFA.SP_GapLeft;
      L     #Ma.FromBCFA1.RV_SP_GapLeft;
      <>I;
      JC    M019;
      T     #Ma.Par.CopyData.SP_GapLeft;
// --Value2
M019: L     #Ma.Par.CopyData.SP_GapRight;
      L     #Ma.ToBCFA.SP_GapRight;
      <>I;
      AN    #Ma.CmdNewJob;
      JC    M020;
      L     0;
M020: T     #tmpSendData.SP_GAP_RIGHT;
      L     #Ma.ToBCFA.SP_GapRight;
      L     #Ma.FromBCFA1.RV_SP_GapRight;
      <>I;
//      AN    #Ma.CmdNewJob               // 1.2
      JC    M025;
      T     #Ma.Par.CopyData.SP_GapRight;
// --Value3
M025: L     #Ma.Par.CopyData.SP_TempRoll;
      L     #Ma.ToBCFA.SP_TempRoll;
      <>I;
      AN    #Ma.CmdNewJob;
      JC    M026;
      L     0;
M026: T     #tmpSendData.SP_TEMP_ROLL;
      L     #Ma.ToBCFA.SP_TempRoll;
      L     #Ma.FromBCFA1.RV_SP_TempRoll;
      <>I;
      JC    M021;
      T     #Ma.Par.CopyData.SP_TempRoll;
// --Value4
M021: L     #Ma.Par.CopyData.SP_FE_RollSpeed;
      L     #Ma.ToBCFA.SP_FE_RollSpeed;
      <>I;
      AN    #Ma.CmdNewJob;
      JC    M027;
      L     0;
M027: T     #tmpSendData.SP_FE_ROLL_SPEED;
      L     #Ma.ToBCFA.SP_FE_RollSpeed;
      L     #Ma.FromBCFA1.RV_SP_FE_RollSpeed;
      <>I;
      JC    M022;
      T     #Ma.Par.CopyData.SP_FE_RollSpeed;
// --Value5
M022: L     #Ma.Par.CopyData.SP_FE_VibroSpeed;
      L     #Ma.ToBCFA.SP_FE_VibroSpeed;
      <>I;
      AN    #Ma.CmdNewJob;
      JC    M023;
      L     0;
M023: T     #tmpSendData.SP_FE_VIBRO_SPEED;
      L     #Ma.ToBCFA.SP_FE_VibroSpeed;
      L     #Ma.FromBCFA1.RV_SP_FE_VibroSpeed;
      <>I;
      JC    M024;
      T     #Ma.Par.CopyData.SP_FE_VibroSpeed;
// --Value6
M024: L     #Ma.Par.CopyData.SP_RC_Option;
      L     #Ma.ToBCFA.SP_RC_Option;
      <>I;
      AN    #Ma.CmdNewJob;
      JC    M028;
      L     0;
M028: T     #tmpSendData.SP_RC_OPTION;
      L     #Ma.ToBCFA.SP_RC_Option;
      L     #Ma.FromBCFA1.RV_SP_RC_Option;
      <>I;
      JC    M029;
      T     #Ma.Par.CopyData.SP_RC_Option;
M029: NOP   0;
//---------------------------
// Send to Hardware
//---------------------------
      A     #Ma.InSimulation;
      JC    M010;
      CALL  "SIEMENS_DPWR_DAT" (
           LADDR                    := #tmpAddr1,
           RECORD                   := #tmpSendData,
           RET_VAL                  := #tmpReturn2);
      L     #tmpReturn2;
      L     0;
      <>I;
      =     #Ma.Par.OutHelpFlags.OutComFaultSend;
      JU    M011;
//---------------------------
// Send to Simulation
//---------------------------
M010: R     #Ma.Par.OutHelpFlags.OutComFaultSend;
      A     "GCS7_Gr_SimDPtoImage";
      L     P#Q 0.0;
      JC    M031;
      OPN   "TEST_IOSimuliOutput";
      L     P#DBX 0.0;
M031: L     #Ma.Par.ParIOByteNr;
      SLD   3;
      +D;
      T     LD 6;	//->Src.BitAddress 
      L     W#16#1002;	//S7 word
      T     LW 0;	//->Src.type
      L     32;	//Length in byte
      T     LW 2;	//->Src.factor
      L     DBNO;
      A     "GCS7_Gr_SimDPtoImage";
      JC    M030;
      L     0;
M030: T     LW 4;	//->Src.DB
      CALL  "SIEMENS_BLKMOV" (
           SRCBLK                   := #tmpSendData,
           RET_VAL                  := #error,
           DSTBLK                   := #Src);
M011: NOP   0;
NETWORK
TITLE = State Code
      L     1;	//Code: StStopped
      A     #Ma.StStopped;
      JC    STC1;
      L     2;	//Code: StStarting
      A     #Ma.StStarting;
      JC    STC1;
      L     3;	//Code: StStandby
      A     #Ma.StStandby;
      JC    STC1;
      L     4;	//Code: StProduction
      A     #Ma.StProduction;
      JC    STC1;
      L     5;	//Code: StStopping
      A     #Ma.StStopping;
      JC    STC1;
      L     6;	//Code: StCalibation
      A     #Ma.StService;
      JC    STC1;
      A     #tmpLocal;
      L     31;	//Code: StFaultCom.Local
      JC    STC;
      L     32;	//Code: StFaultCom.Active
      JC    STC;
STC1: AN    #Ma.OutFaulted;
      JC    STCW;
      +     20;	//StXxxx.Faulted
      JU    STC;
STCW: AN    #Ma.OutWarning;
      JC    STC;
      +     10;	//StXxxx.Warning
STC:  L     #Ma.StCode;	//Old state code
      TAK;
      T     #Ma.StCode;	//Save state code
      <>I;
      L     3;	//Load code for CBit methode
      CC    "SYS_CBitCtrl";
NETWORK
TITLE = Call Motor1
      A     #Ma.FromBCFA2.Sta_MM_1_On;
      =     #Motor1.InpRunFwd;
      A     #Ma.FromBCFA2.Sta_MM_1_Fault;
      =     #Motor1.InpFaultDev;
      NOT;
      =     #Motor1.InLocal;
      SET;
      S     #Motor1.Par.ParLogOff;
      CALL  #Motor1;
NETWORK
TITLE = Call Motor2
      A     #Ma.FromBCFA2.Sta_MM_2_On;
      =     #Motor2.InpRunFwd;
      A     #Ma.FromBCFA2.Sta_MM_2_Fault;
      =     #Motor2.InpFaultDev;
      NOT;
      =     #Motor2.InLocal;
      SET;
      S     #Motor2.Par.ParLogOff;
      CALL  #Motor2;
NETWORK
TITLE = Call Hydraulic
      A     #Ma.FromBCFA2.Sta_HD_On;
      =     #Hydraulic.InpRunFwd;
      A     #Ma.FromBCFA2.Sta_HD_Fault;
      =     #Hydraulic.InpFaultDev;
      NOT;
      =     #Hydraulic.InLocal;
      SET;
      S     #Hydraulic.Par.ParLogOff;
      CALL  #Hydraulic;
NETWORK
TITLE = Call Cooler
      A     #Ma.FromBCFA2.Sta_RC_On;
      =     #Cooler.InpRunFwd;
      A     #Ma.FromBCFA2.Sta_RC_Fault;
      =     #Cooler.InpFaultDev;
      NOT;
      =     #Cooler.InLocal;
      SET;
      S     #Cooler.Par.ParLogOff;
      CALL  #Cooler;
NETWORK
TITLE = Call Engaged
      A     #Ma.FromBCFA2.Sta_Engaged_On;
      =     #Engaged.InpRunFwd;
      A     #Ma.FromBCFA2.Sta_Engaged_Fault;
      =     #Engaged.InpFaultDev;
      NOT;
      =     #Engaged.InLocal;
      SET;
      S     #Engaged.Par.ParLogOff;
      CALL  #Engaged;
NETWORK
TITLE = Call Feeder
      A     #Ma.FromBCFA2.Sta_ROLL_On;
      =     #RollFeeder.InpRunFwd;
      A     #Ma.FromBCFA2.Sta_ROLL_Fault;
      =     #RollFeeder.InpFaultDev;
      NOT;
      =     #RollFeeder.InLocal;
      SET;
      S     #RollFeeder.Par.ParLogOff;
      CALL  #RollFeeder;
NETWORK
TITLE = Call Vibro
      A     #Ma.FromBCFA2.Sta_Vibro_On;	//[1.1]
      =     #VibroFeeder.InpRunFwd;
      A     #Ma.FromBCFA2.Sta_Vibro_Fault;	//[1.1]
      =     #VibroFeeder.InpFaultDev;
      NOT;
      =     #VibroFeeder.InLocal;
      SET;
      S     #VibroFeeder.Par.ParLogOff;
      CALL  #VibroFeeder;
NETWORK
TITLE = Call Flap
      A     #Ma.FromBCFA2.Sta_Flap_Production;
      =     #Flap.InpHN;
      NOT;
      =     #Flap.InpLN;
      A     #Ma.FromBCFA2.Sta_Flap_Fault;
      =     #Flap.InpFaultDev;
      NOT;
      =     #Flap.InLocal;
      SET;
      S     #Flap.Par.ParLogOff;
      CALL  #Flap;
NETWORK
TITLE = Call ProductFlow
      A     #Ma.FromBCFA2.Sta_Flow_Ok;
      =     #ProductFlow.InpTrue;
      A     #Ma.FromBCFA2.Sta_Flow_Fault;
      =     #ProductFlow.InpFaultDev;
      NOT;
      =     #ProductFlow.InLocal;
      SET;
      S     #ProductFlow.Par.ParLogOff;
      CALL  #ProductFlow;
END_FUNCTION_BLOCK

FUNCTION_BLOCK "GCS7_M_DischargerMZAx"	// FB 59
TITLE = Bin discharger with MZAF
//  
//COPYRIGHT:    (C) 1997  BUHLER AG, CH-9240 UZWIL,  SWITZERLAND
//
//PRODUCT:      GCS7
//
//TITLE:        FB 59 Machine Control:Bin discharger with MZAF 
//              MZAF, LL and LS
//
//-------------------------------------------------------------------------
//
//IDENT:        AUTHOR:             DEPT:                       DATE:
//
//FB59.4.0      A. Egli             CT3                         17-Jun-2002
//              New Release with one block 
//FB59.3.1      E.Hanselmann/A.Egli MU664/CT3                   29-Jan-2001
//              Condition for Ma.OutEmpty corrected 
//FB59.3.0      A. Egli             CT3                         11-Oct-1999
//              Local data reduced 
//FB59.2B       K. Tischer          MU664                       06-Mrz-1999
//              CC FC2 not UC FC2
//FB59.2A       A. Egli             CT3                         04-Mai-1998
//              StFault = StCode 32
//FB59.1A       A.Egli              AEE61                       12-Nov-1997
//              1st Release in S7
//
//-------------------------------------------------------------------------
//
//PURPOSE:      MANUAL : see [LL.MA.MZAxxMAN]
//
//RESTRICTIONS: S7
//              ACCU2: Pointer to dynamic datas of the machine
//              ACCU1: Pointer to parameter datas of the machine
//
//-------------------------------------------------------------------------
//
//
AUTHOR : EA
FAMILY : GCS7LL
NAME : MA_MZAF
VERSION : 4.0
VAR
  Ma : UDT 20590;
  MZAF : FB 32;	//Element
  LS : FB 14;	//Element
END_VAR
VAR_TEMP
  tmpFaultStop : BOOL ;
  tmpFaultSum : BOOL ;
  tmpNext : BOOL ;
  tmpEnable : BOOL ;
  tmpEmpty : BOOL ;
  tmpLenDyn : INT ;
END_VAR
BEGIN
NETWORK
TITLE =
      L     16;
      T     #tmpLenDyn;
NETWORK
TITLE = PC Control
//=== Test Object number =====================
      L     "SYS_DirectCtrlDB".PC.ObjectNo;	//PCControl.ObjectNo
      L     #Ma.Par.ParObjectNo;	//Input ObjectNo
      <>I;
      JC    aEnd;
//=== Test OType      ========================
      L     2059;	//Input object type
      L     "SYS_DirectCtrlDB".PC.ObjectType;	//PCControl.ObjectType
      <>I;
      JC    aEnd;
//=== Test Handshake =========================
      A     "SYS_DirectCtrlDB".PC.Hsk.FExamine;	// Handshake.FExamine
      JC    aExa;
      A     "SYS_DirectCtrlDB".PC.Hsk.FDefineCmd;	// Handshake.FDefineCmd
      O     "SYS_DirectCtrlDB".PC.Hsk.FDefinePara;	// Handshake.FDefinePara
      JC    aCmd;
aIni: L     2;	// FcInit
      UC    "SYS_DirectCtrl";
      JU    aEnd;
// Write new commands from PC to Interface of group 
aCmd: A     "SYS_DirectCtrlDB".PC.Cmd1[8];	//Cmd1[8]=CmdOff
      S     #Ma.CmdOff;
      A     "SYS_DirectCtrlDB".PC.Cmd1[9];	//Cmd1[9]=CmdOn
      S     #Ma.CmdOn;
      A     "SYS_DirectCtrlDB".PC.Cmd1[10];	//Cmd1[10]=CmdNext
      S     #Ma.CmdNext;
      A     "SYS_DirectCtrlDB".PC.Cmd1[11];	//Cmd1[11]=CmdFaultReset
      S     #Ma.CmdFaultReset;
      A     "SYS_DirectCtrlDB".PC.Cmd1[13];	//Cmd1[13]=CmdManualOn
      S     #Ma.InManual;
      A     "SYS_DirectCtrlDB".PC.Cmd2[13];	//Cmd1[13]=CmdManualOff
      R     #Ma.InManual;
      A     "SYS_DirectCtrlDB".PC.Cmd1[1];	//Cmd1[1]=CmdRestDischargeOn
      S     #Ma.InRestDischarge;
      A     "SYS_DirectCtrlDB".PC.Cmd2[1];	//Cmd2[1]=CmdRestDischargeOff
      R     #Ma.InRestDischarge;
      JU    aIni;
aExa: TAR2;	// Address Dynamic data
      T     "SYS_DirectCtrlDB".GC.InDynAddr;	// -->PCControl.GC.InDynAddr
      L     #tmpLenDyn;	// Length Dynamic data
      T     "SYS_DirectCtrlDB".GC.InDynLen;	// -->PCControl.GC.InDynLen
      L     0;
      T     "SYS_DirectCtrlDB".GC.InParaAddr;	// -->PCControl.GC.InParaAddr
      T     "SYS_DirectCtrlDB".GC.InParaLen;	// -->PCControl.GC.InParaLen
      L     1;	// Code FcExamine
      UC    "SYS_DirectCtrl";
      L     10;	//Revision
      T     "SYS_DirectCtrlDB".GC.Revision;
aEnd: NOP   0;
NETWORK
TITLE = Interlocking
//===Global Group Orders===
      A     "GCS7_Gr_OutManualOn";	//Gr.OutManualOn
      S     #Ma.InManual;
      A     "GCS7_Gr_OutManualOff";	//Gr.OutManualOff
      R     #Ma.InManual;
      A     #Ma.InManual;
      S     "GCS7_Gr_InManual";	//Gr.InManual
      A     #Ma.CmdNext;
      AN    #Ma.InManual;
      O     #Ma.CmdOn;
      =     #tmpNext;
      A     #Ma.InManual;
      ON    #Ma.InLocal;
      A     #Ma.InEnable;
      AN    #Ma.CmdOff;
      =     #tmpEnable;
//---- Low level 
      A     #Ma.InUncovered;
      ON    #Ma.Par.ParWithLL;
      A(;
      O     #LS.StFalse;
      O     #LS.StCtoTrue;	//[3.1]old=#LS.StCtoFalse
      );
      S     #Ma.OutEmpty;
      A     #LS.StTrue;
      AN    #Ma.Par.ParWithLL;
      O     #Ma.InCovered;
      R     #Ma.OutEmpty;
      A     #Ma.OutEmpty;
      AN    #Ma.InRestDischarge;
      A     #Ma.Par.ParWithLL;
      =     #tmpEmpty;
//--- Fault----
      A     #LS.StFault;
      O     #MZAF.StFault;
      =     #tmpFaultSum;
// 
//--- Interlocking MZAF
      A     #Ma.StWaiting;
      AN    #Ma.InLocal;
      AN    #Ma.InManual;
      O     #tmpNext;
      S     #MZAF.CmdNext;
      S     #MZAF.InEnable;
      A     #tmpEmpty;
      AN    #Ma.InRestDischarge;
      AN    #Ma.InManual;
      ON    #tmpEnable;
      O     #tmpFaultSum;
      R     #MZAF.InEnable;
//New job 
      A     #Ma.CmdNewJob;
      S     #MZAF.CmdNewJob;
// 
//--- Local mode --
      A     #Ma.InLocal;
      AN    #Ma.InManual;
      =     #MZAF.InLocal;
      =     #LS.InLocal;
//--- Fault Reset -------------
      A     #Ma.CmdFaultReset;
      S     #MZAF.CmdFaultReset;
      S     #LS.CmdFaultReset;
// 
//--- Monitoring LS
      A     #Ma.InCovered;
      A     #Ma.Par.ParWithLL;
      O     #Ma.InMonLSFault;
      A     #MZAF.StStarted;
      AN    #Ma.InManual;
      =     #LS.InMonTrue;
      SET;
      R     #LS.InMonFalse;
NETWORK
TITLE = Call MZAF
      CALL  #MZAF;
NETWORK
TITLE = Call Digital Input: LS
      CALL  #LS;
NETWORK
TITLE = Jump to actual state
      A     #Ma.StStopped;
      JC    S0;	// ===> State
      A     #Ma.StStarted;
      JC    S2;	// ===> State
      A     #Ma.StStarting;
      JC    S1;	// ===> State
      A     #Ma.StStopping;
      JC    S3;	// ===> State
      A     #Ma.StFault;
      JC    S4;	// ===> State
      A     #Ma.StWaiting;
      JC    S5;	// ===> State
NETWORK
TITLE = Stopped
//any Transition 
xxS0: S     #Ma.StStopped;	// ===> Initialisation
//=== Logic
// Condition for StFault
S0:   A     #tmpFaultSum;
      R     #Ma.StStopped;
      JC    xxS4;	//--> ST_FAULT:
// Condition for StStarting
      AN    #MZAF.StStopped;
      R     #Ma.StStopped;
      JC    xxS1;	//--> StStarting
// Condition for StWaiting
      A     #tmpNext;
      A     #tmpEnable;
      A     #tmpEmpty;
      AN    #Ma.InRestDischarge;
      R     #Ma.StStopped;
      JC    xxS5;	//--> StWaiting
      JU    OUT;
NETWORK
TITLE = StStarting
//any Transition 
xxS1: S     #Ma.StStarting;
//=== Logic
// Condition for StFault
S1:   A     #tmpFaultSum;
      R     #Ma.StStarting;
      JC    xxS4;	//--> StFault
// Condition for StStarted
      A     #MZAF.StStarted;
      R     #Ma.StStarting;
      JC    xxS2;	//-->StStarted
// Condition for StStopping
      AN    #MZAF.StAdjusting;
      R     #Ma.StStarting;
      JC    xxS3;	//-->StStopping
      JU    OUT;
NETWORK
TITLE = StStarted
//any Transition 
xxS2: S     #Ma.StStarted;
//=== Logic
// Condition for StFault
S2:   A     #tmpFaultSum;
      R     #Ma.StStarted;
      JC    xxS4;	//--> StFault
// Condition for StWaiting
      A     #tmpEmpty;
      AN    #Ma.InRestDischarge;
      AN    #MZAF.StStarted;
      AN    #MZAF.StAdjusting;
      R     #Ma.StStarted;
      JC    xxS5;	//-->StWaiting
// Condition for StStopping
      AN    #MZAF.StStarted;
      AN    #MZAF.StAdjusting;
      R     #Ma.StStarted;
      JC    xxS3;	//-->StStopping
      JU    OUT;
NETWORK
TITLE = Stopping
//any Transition 
xxS3: S     #Ma.StStopping;
//=== Logic
// Condition for StFault
S3:   A     #tmpFaultSum;
      R     #Ma.StStopping;
      JC    xxS4;	//--> StFault
// Condition for StStopped
      A     #MZAF.StStopped;
      R     #Ma.StStopping;
      JC    xxS0;	//-->StStopped
// Condition for StStarting
      A     #MZAF.StStarted;
      R     #Ma.StStopping;
      JC    xxS1;	//-->StStarting
      JU    OUT;
NETWORK
TITLE = Fault
//any Transition 
xxS4: S     #Ma.StFault;
      JU    OUT;
//=== Logic
S4:   A     #tmpFaultSum;
      JC    OUT;
//---- Transition --
      R     #Ma.StFault;
      JU    xxS0;	//-->StStopping 
NETWORK
TITLE = StWaiting
//any Transition 
xxS5: S     #Ma.StWaiting;
      JU    OUT;
//=== Logic
// Condition for StFault
S5:   A     #tmpFaultSum;
      R     #Ma.StWaiting;
      JC    xxS4;	//--> StFault
// Condition for StStarted
      A     #MZAF.StStarted;
      R     #Ma.StWaiting;
      JC    xxS2;	//-->StStarted
// Condition for StStopping
      AN    #tmpEnable;
      R     #Ma.StWaiting;
      JC    xxS3;	//-->StStopping
      JU    OUT;
NETWORK
TITLE = State Code
// State     StCode
// ----------------------
// StFault32
// StStopped    1
// StStarting   2
// StWaiting    3
// StStarted    4
// StStopping  7
OUT:  A     #Ma.StStopped;
      L     1;	//Code=StStopped
      JC    Code;
      A     #Ma.StWaiting;
      L     3;	//Code=StWaiting
      JC    Code;
      A     #Ma.StStarted;
      L     4;	//Code=StStarted
      JC    Code;
      A     #Ma.StStarting;
      L     2;	//Code=StStarting
      JC    Code;
      A     #Ma.StStopping;
      L     7;	//Code=StStopping 
      JC    Code;
      L     32;	//Code=StFault 
Code: L     #Ma.StCode;	// Old state code
      TAK;
      T     #Ma.StCode;	// Save state code
      <>I;
      L     3;
      CC    "SYS_CBitCtrl";	//Set change bit
NETWORK
TITLE = Global End
      CLR;	//---Clear all commands
      =     #Ma.CmdOn;
      =     #Ma.CmdOff;
      =     #Ma.CmdNext;
      =     #Ma.CmdFaultReset;
      =     #Ma.CmdNewJob;
END_FUNCTION_BLOCK

FUNCTION_BLOCK "GCS7_M_Aspiration"	// FB 60
TITLE = Aspiration Fan with 1 Airlock
//  
//COPYRIGHT:    (C) 1997  BUHLER AG, CH-9240 UZWIL, SWITZERLAND
//
//PRODUCT:      GCS7
//
//TITLE:        FB 60 Machine Control:Aspiration  
//
//REVISION:     10
//-------------------------------------------------------------------------
//
//IDENT:        AUTHOR:             DEPT:                       DATE:
//
//FB60.5.13     M. Miotto           MU93                        13-Nov-2008
//              - Condition StStarted if Discharger is off during startup
//FB60.5.12     A. Egli             CT3                         21-Aug-2008
//              - ARF: InEnableHN only if Fan is started (MAUB)
//              - ARF: InEnableLN only if Fan is stopped (MAUA)
//FB60.5.11     A. Egli             CT3                         09-Apr-2008
//              - InDisableDischarger added
//              - ARF: Interlocking with Fan.OutpRunFwd
//FB60.5.10     G. Shingler         CDDP                        22-Sep-2006
//              InDisableFilter added
//FB60.5.9      A.Egli              CT3                         25-Jan-2005
//              Transition StStarted to StStopping, when no element is started
//FB60.5.8      A.Egli              CT3                         22-Jun-2004
//              Use HLAirlock.OutTimeoutTime in Transition to StStarted
//              Undo change [5.4]
//FB60.5.7      A.Egli              CT3                         27-Mai-2004
//              Undo changes of [5.6]
//FB60.5.6      K.Tischer           CT3                         12-Feb-2004
//              after inDisableAirlock Ma.stStarting
//FB60.5.5      K.Tischer           CT3                         10-Feb-2004
//              #ARF.InEnableHN   new:#Fan.StStartedFwd (old:#Fan.OutpRunFwd)  
//FB60.5.4      A.Egli              CT3                         11-Nov-2003
//              Continue StStarted --> StStopping when Airlock is stopped
//FB60.5.3      A.Egli              CT3                         01-Okt-2003
//              Continue running Filter if InDisableAirlock
//FB60.5.2      A. Egli             CT3                         18-Aug-2003
//              Condition for Idling
//FB60.5.1      A. Egli             CT3                         22-Jul-2003
//              Filter.InLocal
//FB60.5.0      A. Egli             CT3                         17-Dec-2002
//              New Release with one block
//FB60.4.4      P.Engler            CT3                         17-Dec-2002
//              Run filter if InDisableAirlock
//FB60.4.3      A. Egli             CT3                         25-Sep-2001
//              ARF.StHN as contion for transition -->StStarted
//FB60.4.2      A. Egli             CT3                         24-Aug-2000
//              Condition for InLocal
//FB60.4.1      A. Egli             CT3                         27-Jun-2000
//              Monitoring HL Airlock always 
//FB60.4.0      A. Egli             CT3                         25-Mai-2000
//              New Element Discharger 
//FB60.3.3      A. Egli             CT3                         24-Jan-2000
//              -Condition StStopping to StStarting
//              -Pressure.InPrealarmTrue
//FB60.3.2      A. Egli             CT3                         24-Jan-2000
//              Condition StStarting to StStopping
//FB60.3.1      A. Egli             CT3                         15-Nov-1999
//              Monitoring HLAirLock adapted
//FB60.3.0      A. Egli             CT3                         11-Oct-1999
//              Local data reduced
//FB60.2C       A. Egli             CT3                         17-Aug-1999
//              No interlocking and with filter door
//FB60.2B       K. Tischer          MU664                       06-Mrz-1999
//              CC FC2 not UC FC2
//FB60.2A       A. Egli             CT3                         04-Mai-1998
//              StFault = StCode 32
//FB60.1A       A.Egli              AEE61                       8-Jul-1997
//              1st Release in S7
//
//-------------------------------------------------------------------------
//
//PURPOSE:      MANUAL : see [LL.ASAxxMAN]
//
//RESTRICTIONS: S7
//
//-------------------------------------------------------------------------
//
//
AUTHOR : EA
FAMILY : GCS7LL
NAME : Aspirati
VERSION : 5.13
VAR
  Ma : UDT 20600;
  Airlock : FB 12;	//Elememt airlock
  Fan : FB 12;	//Elememt Fan
  Filter : FB 11;	//Elememt Filter control
  ARF : FB 13;	//Elememt Air regulation flap
  LSDoor : FB 14;	//Element filter door
  Pressure : FB 14;	//Element Filter Pressure
  HLAirlock : FB 14;	//Elememt HL Airlock
  Discharger : FB 12;	//Elememt Discharger (Vibro)
END_VAR
VAR_TEMP
  tmpFaultStop : BOOL ;
  tmpFaultSum : BOOL ;
  tmpLocal : BOOL ;
  tmpNext : BOOL ;
  tmpEnableVibro : BOOL ;
  tmpPulsingMode : BOOL ;
  tmpLenDyn : INT ;
END_VAR
BEGIN
NETWORK
TITLE =
      L     20;
      T     #tmpLenDyn;
NETWORK
TITLE = PC Control
//=== Test Object number =====================
      L     "SYS_DirectCtrlDB".PC.ObjectNo;	//PCControl.ObjectNo
      L     #Ma.Par.ParObjectNo;	//Input ObjectNo
      <>I;
      JC    aEnd;
//=== Test OType      ========================
      L     2060;	//Input object type
      L     "SYS_DirectCtrlDB".PC.ObjectType;	//PCControl.ObjectType
      <>I;
      JC    aEnd;
//=== Test Handshake =========================
      A     "SYS_DirectCtrlDB".PC.Hsk.FExamine;	// Handshake.FExamine
      JC    aExa;
      A     "SYS_DirectCtrlDB".PC.Hsk.FDefineCmd;	// Handshake.FDefineCmd
      JC    aCmd;
      A     "SYS_DirectCtrlDB".PC.Hsk.FDefinePara;	// Handshake.FDefinePara
      JC    aPar;
aIni: L     2;	// FcInit
      UC    "SYS_DirectCtrl";
      JU    aEnd;
// Write parameter 
aPar: LAR1  P#DBX 58.0;
      L     P#6.0;
      +AR1;
      L     DBW [AR1,P#4.0];
      T     #Ma.Par.ParVibroOnTime;
      L     DBW [AR1,P#6.0];
      T     #Ma.Par.ParVibroOffTime;
// Write new commands from PC to Interface of group 
aCmd: A     "SYS_DirectCtrlDB".PC.Cmd1[8];	//Cmd1[8]=CmdOff
      S     #Ma.CmdOffMan;
      A     "SYS_DirectCtrlDB".PC.Cmd1[9];	//Cmd1[9]=CmdOn
      S     #Ma.CmdOnMan;
      A     "SYS_DirectCtrlDB".PC.Cmd1[10];	//Cmd1[10]=CmdNext
      S     #Ma.CmdNext;
      A     "SYS_DirectCtrlDB".PC.Cmd1[11];	//Cmd1[11]=CmdFaultReset
      S     #Ma.CmdFaultReset;
      A     "SYS_DirectCtrlDB".PC.Cmd1[13];	//Cmd1[13]=CmdManualOn
      S     #Ma.InManual;
      A     "SYS_DirectCtrlDB".PC.Cmd2[13];	//Cmd2[13]=CmdManualOff
      R     #Ma.InManual;
      A     "SYS_DirectCtrlDB".PC.Cmd1[14];	//Cmd1[14]=CmdFanOffMan
      S     #Ma.CmdFanOffMan;
      AN    "SYS_DirectCtrlDB".PC.Hsk.FDefineCmd;	// Handshake.FDefineCmd
      JC    aIni;
      JU    aIni;
aExa: TAR2;	// Address dynamic data
      T     "SYS_DirectCtrlDB".GC.InDynAddr;	// -->PCControl.GC.InDynAddr
      L     #tmpLenDyn;	// Length Dynamic data
      T     "SYS_DirectCtrlDB".GC.InDynLen;	// -->PCControl.GC.InDynLen
      L     0;
      T     "SYS_DirectCtrlDB".GC.InParaAddr;	// -->PCControl.GC.InParaAddr
      T     "SYS_DirectCtrlDB".GC.InParaLen;	// -->PCControl.GC.InParaLen
      L     1;	// Code FcExamine
      UC    "SYS_DirectCtrl";
      L     10;	//Revision
      T     "SYS_DirectCtrlDB".GC.Revision;
aEnd: NOP   0;
NETWORK
TITLE = Pulsing mode Discharger
      L     #Ma.Par.ParVibroOffTime;
      L     0;
      <>I;
      A(;
      L     #Ma.Par.ParVibroOffTime;
      <>I;
      );
      =     #tmpPulsingMode;
NETWORK
TITLE = Interlocking
//===Global Group Orders===
      A     "GCS7_Gr_OutManualOn";	//Gr.OutManualOn
      S     #Ma.InManual;
      A     "GCS7_Gr_OutManualOff";	//Gr.OutManualOff
      R     #Ma.InManual;
      A     #Ma.InManual;
      S     "GCS7_Gr_InManual";	//Gr.InManual
      A     #Ma.CmdNext;
      AN    #Ma.InManual;
      O     #Ma.CmdOnMan;
      =     #tmpNext;
      A     #Ma.InLocal;
      AN    #Ma.InManual;
      =     #tmpLocal;
//--- Fault----
      A     #Discharger.StFault;
      A     #Ma.Par.ParWithDischarger;
      O     #LSDoor.StFault;
      O     #Pressure.StFault;
      O     #Airlock.StFault;
      O     #Fan.StFault;
      O     #ARF.StFault;
      O     #Filter.StFault;
      O     #HLAirlock.StFault;
      =     #tmpFaultSum;
// 
//--- Interlocking airlock 
      A     #LSDoor.StTrue;
      ON    #Ma.Par.ParWithLSDoor;
      AN    #Ma.CmdOffMan;
      AN    #Ma.InDisableAirlock;
      =     #Airlock.InEnableFwd;
      A     #tmpNext;
      A     #Ma.InEnable;
      S     #Airlock.CmdNext;
      AN    #Fan.StStartedFwd;
      ON    #Ma.Par.ParWithFan;
      A     #Ma.InSeqStop;
      AN    #Ma.InManual;
      ON    #Ma.InEnable;
      =     #Airlock.InSeqStop;
//--- Interlocking Filter 
      =     #Filter.InSeqStop;
      A     #Airlock.StStartedFwd;
      ON    #Ma.Par.ParWithAirlock;
      A     #Airlock.InEnableFwd;	//[3.3]
      O(;	//[4.4]
      AN    #Ma.InDisableAirlock;	//[4.4]
      O     #Ma.InEnable;	//[4.4]
      A(;	//[5.3]
      A     #HLAirlock.StFalse;	//[5.3]
      O     #HLAirlock.StCtoTrue;	//[5.3]
      A     #Ma.Par.ParWithHLAirlock;	//[5.3]
      O     #Ma.Par.ParWithDischarger;	//[5.3]
      );	//[5.3]
      );
      AN    #Ma.InDisableFilter;	//[5.10]
      =     #Filter.InEnable;
      A     #Airlock.StStartedFwd;
      ON    #Ma.Par.ParWithAirlock;	//[4.4]
      A(;	//[4.4]
      A     #Discharger.StStartedFwd;	//[4.4]
      O     #Ma.InDisableDischarger;	//[5.13]
      ON    #Ma.Par.ParWithDischarger;	//[4.4]
      O     #tmpPulsingMode;	//[5.0]
      );	//[4.4]
      O     #Ma.InDisableAirlock;	//[4.4]
      A     #tmpNext;	//[4.4]
      S     #Filter.CmdNext;
// 
//--- Interlocking Fan
//2C: U     #LSDoor.StTrue;
//2C: ON    #Ma.Par.ParWithLSDoor;
      A     #Ma.InEnable;
      AN    #Ma.CmdFanOffMan;
      AN    #Ma.CmdOffMan;
      =     #Fan.InEnableFwd;
      A     #ARF.StLN;
      ON    #Ma.Par.ParWithARF;
      A(;	//[4.4]
      A     #Ma.InDisableAirlock;	//[4.4]
      A     #Ma.Par.ParWithDischarger;	//[4.4]
      O     #Filter.StStarted;	//[4.4]
      O     #Ma.InDisableFilter;	//[5.10]
      ON    #Ma.Par.ParWithFilter;	//[4.4]
      );
      A(;
      A     #Airlock.StStartedFwd;
      ON    #Ma.Par.ParWithAirlock;
      O     #Ma.InDisableAirlock;	//[4.4]
      );
      A(;
      A     #Discharger.StStartedFwd;	//[4.4]
      O     #Ma.InDisableDischarger;	//[5.13]
      ON    #Ma.Par.ParWithDischarger;	//[4.4]
      O     #Ma.InDisableAirlock;	//[4.4]
      O     #tmpPulsingMode;	//[5.0]
      );
      A     #tmpNext;
      S     #Fan.CmdNext;
// 
      A     #Ma.InSeqStop;
      AN    #Ma.InManual;
      =     #Fan.InSeqStop;
//--- Interlocking ARF
      A     #Fan.StStartedFwd;	//[5.5] MAUB=Command to open flap ,MAUA=Command to monitoring open position
      =     #ARF.InEnableHN;
      A     #Fan.StStopped;	//[5.5]
      O     #Fan.StFault;	//[5.11][5.12](MAUA)
      =     #ARF.InEnableLN;	//MAUB=Command to close flap ,MAUA=Command to monitoring closed position
      SET;
      S     #ARF.CmdNext;
      AN    #Ma.Par.ParWithDischarger;
      JC    InX1;
      A     #Ma.StStarted;	//5.0
      A     #tmpPulsingMode;	//5.0
      O     #tmpNext;	//5.0
      A     #Discharger.InEnableFwd;	//[5.11]
      S     #Discharger.CmdNext;
// 
//--- Interlocking LSDoore 
InX1: SET;
      =     #LSDoor.InMonTrue;
// 
//--- Interlocking pressure 
      A     #Ma.InEnable;
      AN    #tmpLocal;
      O     #Ma.InManual;
      AN    #Ma.Par.ParWithFan;
      O     #Fan.StStartedFwd;	// [4.0] 
      =     #Pressure.InMonTrue;
      =     #Pressure.InPreAlarmTrue;	//[3.3] 
// 
//--- Interlocking HL 
//      U     #Airlock.StStartedFwd;      //3.1 
//      O     #Ma.InDisableAirlock;   //3.1
      SET;	//4.1
      =     #HLAirlock.InMonFalse;
//--- Local mode --
      A(;
      A     #Fan.StStopped;
      ON    #Ma.Par.ParWithFan;
      );
      A(;
      A     #Airlock.StStopped;
      ON    #Ma.Par.ParWithAirlock;
      );
      A     #tmpLocal;
      =     #LSDoor.InLocal;	//[4.2]
      =     #Pressure.InLocal;	//[4.2]
      A     #tmpLocal;
      =     #Fan.InLocal;
      =     #ARF.InLocal;
      =     #HLAirlock.InLocal;
      =     #Airlock.InLocal;
      =     #Filter.InLocal;	//[5.1]
      AN    #Ma.Par.ParWithDischarger;
      JC    InL1;
      A     #tmpLocal;
      =     #Discharger.InLocal;
//--- Fault Reset -------------
InL1: A     #Ma.CmdFaultReset;
      S     #Pressure.CmdFaultReset;
      S     #LSDoor.CmdFaultReset;
      S     #Fan.CmdFaultReset;
      S     #Airlock.CmdFaultReset;
      S     #ARF.CmdFaultReset;
      S     #Filter.CmdFaultReset;
      S     #HLAirlock.CmdFaultReset;
      AN    #Ma.Par.ParWithDischarger;
      JC    InF1;
      A     #Ma.CmdFaultReset;
      S     #Discharger.CmdFaultReset;
//Warning
InF1: AN    #Pressure.StTrue;
      A     #Ma.Par.ParWithPressure;
      O;
      A     #Ma.Par.ParWithFilter;
      A     #Filter.OutWarning;
      =     #Ma.OutWarning;
NETWORK
TITLE = Interlocking Discharger/ Vibro Time (5.0)
      AN    #Ma.Par.ParWithDischarger;
      JC    VBEN;
//== timer Vibro                        
//Start Vibro immediatly at negativ flag of
      A     #Airlock.StStartedFwd;
      ON    #Ma.Par.ParWithAirlock;
      A     #Airlock.InEnableFwd;
      =     #tmpEnableVibro;
//----------------------
//Init Pulsing time
      A     #tmpEnableVibro;
      A     #tmpPulsingMode;
      JC    vtJ1;
      L     0;
      T     #Ma.Par.OutDelayTime;
      S     #Ma.OutPulseVibroOn;
      JU    vtOT;
//----------------------
//Count timer
vtJ1: A     #Ma.OutPulseVibroOn;	//[5.11]
      A     #Ma.InDisableDischarger;	//[5.11]
      ON    "GCS7_Gr_OutTick200ms";	//Gr.OutTick200ms
      JC    vtOT;
      L     #Ma.Par.OutDelayTime;
      +     2;
      T     #Ma.Par.OutDelayTime;
//----------------------
//Vibro off time
      A     #Ma.OutPulseVibroOn;
      JC    vtOn;
      L     #Ma.Par.ParVibroOffTime;
      L     #Ma.Par.OutDelayTime;
      >=I;
      JC    vtOT;
      S     #Ma.OutPulseVibroOn;
      JU    vtJ0;
//----------------------
//Vibro on time
vtOn: L     #Ma.Par.ParVibroOnTime;
      <I;
      JC    vtOT;
      R     #Ma.OutPulseVibroOn;
vtJ0: L     0;
      T     #Ma.Par.OutDelayTime;
//----------------------
//Interlocking Discharger
vtOT: A     #Ma.OutPulseVibroOn;	//[5.0]
      AN    #Ma.InDisableDischarger;	//[5.11]
      A     #tmpEnableVibro;
      =     #Discharger.InEnableFwd;
      A     #Airlock.InSeqStop;
      =     #Discharger.InSeqStop;
VBEN: NOP   0;
NETWORK
TITLE = Call Digital Input: LS Filter Door
      AN    #Ma.Par.ParWithLSDoor;
      JC    el2;
      CALL  #LSDoor;
NETWORK
TITLE = Call Digital Input: Pressure
el2:  AN    #Ma.Par.ParWithPressure;
      JC    el3;
      CALL  #Pressure;
NETWORK
TITLE = Call Fan
el3:  AN    #Ma.Par.ParWithFan;
      JC    el4;
      CALL  #Fan;
NETWORK
TITLE = Call Airlock
el4:  AN    #Ma.Par.ParWithAirlock;
      JC    el5;
      CALL  #Airlock;
NETWORK
TITLE = Call Digital Output: Filter control unit
el5:  AN    #Ma.Par.ParWithFilter;
      JC    el6;
      CALL  #Filter;
NETWORK
TITLE = Call VLS: Air legulation flap
el6:  AN    #Ma.Par.ParWithARF;
      JC    el7;
      CALL  #ARF;
NETWORK
TITLE = Call Digital Input: HLAirlock
el7:  AN    #Ma.Par.ParWithHLAirlock;
      JC    el8;
      CALL  #HLAirlock;
NETWORK
TITLE = Call Discharger
el8:  AN    #Ma.Par.ParWithDischarger;
      JC    el9;
      CALL  #Discharger;
el9:  NOP   0;
NETWORK
TITLE = Jump to actual state
      A     #Ma.StStopped;
      JC    S0;	// ===> State
      A     #Ma.StStarted;
      JC    S2;	// ===> State
      A     #Ma.StStarting;
      JC    S1;	// ===> State
      A     #Ma.StStopping;
      JC    S3;	// ===> State
      A     #Ma.StIdling;
      JC    S5;	// ===> State
      A     #Ma.StFault;
      JC    S4;	// ===> State
NETWORK
TITLE = Stopped
//any Transition 
xxS0: S     #Ma.StStopped;	// ===> Initialisation
      L     1;	// StCode=Stopped
      JU    OUT;
//=== Logic
// Condition for StFault
S0:   A     #tmpFaultSum;
      R     #Ma.StStopped;
      JC    xxS4;	//--> ST_FAULT:
// Condition for StStarting
      AN    #Fan.StStopped;
      A     #Ma.Par.ParWithFan;
      O;
      AN    #Airlock.StStopped;
      A     #Ma.Par.ParWithAirlock;
      O;
      AN    #Filter.StStopped;
      A     #Ma.Par.ParWithFilter;
      R     #Ma.StStopped;
      JC    xxS1;	//--> StStarting
      JU    OUT;
NETWORK
TITLE = StStarting
//any Transition 
xxS1: S     #Ma.StStarting;
      L     2;	// StCode=Starting
      JU    OUT;
//=== Logic
// Condition for StFault
S1:   A     #tmpFaultSum;
      R     #Ma.StStarting;
      JC    xxS4;	//--> StFault
// Condition for StStarted
      A     #Fan.StStartedFwd;
      ON    #Ma.Par.ParWithFan;
      A(;
      A     #Airlock.StStartedFwd;
      O     #Ma.InDisableAirlock;	//[4.4]
      ON    #Ma.Par.ParWithAirlock;
      );
      A(;	//[4.4]
      A     #Discharger.StStartedFwd;	//[4.4]
      O     #Ma.InDisableDischarger;	//[5.13]
      O     #Ma.InDisableAirlock;	//[4.4]
      ON    #Ma.Par.ParWithDischarger;	//[4.4]
      O     #tmpPulsingMode;	//[5.0]
      );	//[4.4]
      A(;	//[4.4]
      A     #Ma.InDisableAirlock;	//[4.4]
      A     #Ma.Par.ParWithDischarger;	//[4.4]
      O     #Ma.InDisableFilter;	//[5.10]
      O     #Filter.StStarted;	//[4.4]
      ON    #Ma.Par.ParWithFilter;	//[4.4]
      );
      A(;	//[3.3]
      AN    #Ma.Par.ParWithHLAirlock;	//[3.3]
      O     #HLAirlock.StFalse;	//[3.3]
      O     #HLAirlock.OutTimeoutTime;	//[5.8]
      );	//[3.3]
      A(;	//[3.3]
      AN    #Ma.Par.ParWithPressure;	//[3.3]
      O     #Pressure.StTrue;	//[3.3]
      );	//[3.3]
      A(;	//[4.3]
      A     #ARF.StHN;	//[4.3]
      ON    #Ma.Par.ParWithARF;	//[4.3]
      );	//[4.3]
      R     #Ma.StStarting;
      JC    xxS2;	//-->StStarted
// Condition for StStopping
      A     #Fan.StStopped;	//[3.2]
      O     #Fan.StStopping;
      ON    #Ma.Par.ParWithFan;
      A(;
      AN    #Airlock.StStarting;
      AN    #Airlock.StStartedFwd;
      ON    #Ma.Par.ParWithAirlock;
      );
      A(;
      AN    #Filter.StStarting;
      AN    #Filter.StStarted;
      ON    #Ma.Par.ParWithFilter;
      );
      R     #Ma.StStarting;
      JC    xxS3;	//-->StStopping
// Condition for StIdling
      A     #Airlock.StStartedFwd;
      A     #Airlock.InSeqStop;
      A     #Ma.Par.ParWithAirlock;
      O;
      A     #Filter.StStarted;
      A     #Filter.InSeqStop;
      AN    #Ma.Par.ParWithAirlock;
      R     #Ma.StStarting;
      JC    xxS5;	//-->StIdling
      JU    OUT;
NETWORK
TITLE = StStarted
//any Transition 
xxS2: S     #Ma.StStarted;
      JU    OUT;
//=== Logic
// Condition for StFault
S2:   A     #tmpFaultSum;
      R     #Ma.StStarted;
      JC    xxS4;	//--> StFault
// Condition for StIdling
      A(;
      A     #Airlock.StStartedFwd;
      A     #Airlock.InSeqStop;
      A     #Ma.Par.ParWithAirlock;
      O;
      A     #Filter.StStarted;
      A     #Filter.InSeqStop;
      AN    #Ma.Par.ParWithAirlock;
      O;
      A     #Filter.StStarted;
      A     #Fan.InSeqStop;
      AN    #Ma.Par.ParWithAirlock;
      O;	//[5.2]
      A     #Fan.InSeqStop;	//[5.2]
      A     #Ma.Par.ParWithFan;	//[5.2]
      );
      A(;
      AN    #Fan.StStartedFwd;
      ON    #Ma.Par.ParWithFan;
      );
      R     #Ma.StStarted;
      JC    xxS5;	//-->StIdling  
// Condition for StStopping
      AN    #Fan.StStartedFwd;
      A     #Ma.Par.ParWithFan;
      O;
      AN    #Airlock.StStartedFwd;
//[5.7]      UN    #Airlock.StStarting         //[5.6]
      AN    #Ma.InDisableAirlock;	//[4.4]
      A     #Ma.Par.ParWithAirlock;
      AN    #Ma.Par.ParWithFan;	//[4.4][5.4][5.8]
      O;
      AN    #Filter.StStarted;	//[4.4]
      AN    #Ma.InDisableAirlock;	//[4.4]
      AN    #Ma.InDisableFilter;	//[5.10]
      A     #Ma.Par.ParWithFilter;	//[4.4]
      AN    #Ma.Par.ParWithFan;	//[4.4][5.4][5.8]
      O;	//[5.9]
      AN    #Fan.StStartedFwd;	//[5.9]
      AN    #Filter.StStarted;	//[5.9]
      AN    #Airlock.StStartedFwd;	//[5.9]
      R     #Ma.StStarted;
      JC    xxS3;	//-->StStopping
      JU    OUT;
NETWORK
TITLE = Stopping
//any Transition 
xxS3: S     #Ma.StStopping;
      JU    OUT;
//=== Logic
// Condition for StFault
S3:   A     #tmpFaultSum;
      R     #Ma.StStopping;
      JC    xxS4;	//--> StFault
// Condition for StStopped
      A     #Filter.StStopped;
      ON    #Ma.Par.ParWithFilter;
      A(;
      A     #Fan.StStopped;
      ON    #Ma.Par.ParWithFan;
      );
      A(;
      A     #Airlock.StStopped;
      ON    #Ma.Par.ParWithAirlock;
      );
      R     #Ma.StStopping;
      JC    xxS0;	//-->StStopped
// Condition for StStarting //[3.3]
      AN    #Fan.StStopped;
      AN    #Fan.StStopping;
      ON    #Ma.Par.ParWithFan;
      A(;
      A     #Airlock.StStarting;
      O     #Airlock.StStartedFwd;
      O     #Ma.InDisableAirlock;	//[4.4]
      ON    #Ma.Par.ParWithAirlock;
      );
      A(;
      A     #Filter.StStarting;
      O     #Filter.StStarted;
      O     #Ma.InDisableAirlock;	//[4.4]
      O     #Ma.InDisableFilter;	//[5.10]
      ON    #Ma.Par.ParWithFilter;
      );
      R     #Ma.StStopping;
      JC    xxS1;	//-->StStarting
      JU    OUT;
NETWORK
TITLE = Fault
//any Transition 
xxS4: S     #Ma.StFault;
      JU    OUT;
//=== Logic
S4:   A     #tmpFaultSum;
      JC    OUT;
//    ---- Transition --
      R     #Ma.StFault;
      JU    xxS0;	//-->StStopping 
NETWORK
TITLE = StIdling
//any Transition 
xxS5: S     #Ma.StIdling;
      JU    OUT;
//=== Logic
// Condition for StFault
S5:   A     #tmpFaultSum;
      R     #Ma.StIdling;
      JC    xxS4;	//-->StFault
// Condition for StStopping
      AN    #Airlock.StStartedFwd;
      A     #Ma.Par.ParWithAirlock;
      O;
      AN    #Filter.StStarted;
      AN    #Ma.Par.ParWithAirlock;
      R     #Ma.StIdling;
      JC    xxS3;	//-->StStopping  
// Condition for StStarted
      AN    #Fan.StStopped;
      AN    #Fan.StStopping;
      A     #Ma.Par.ParWithFan;
      O;
      A     #Airlock.StStartedFwd;
      AN    #Airlock.InSeqStop;
      A     #Ma.Par.ParWithAirlock;
      O;
      A     #Filter.StStarted;
      AN    #Filter.InSeqStop;
      AN    #Ma.Par.ParWithAirlock;
      A     #Ma.Par.ParWithFilter;
      R     #Ma.StIdling;
      JC    xxS1;	//-->StStarting
      JU    OUT;
NETWORK
TITLE = State Code
// State           StCode
// ----------------------
// StFault            32
// StStopped          1
// StStarting         2
// StStarted          3
// StWarning          4
// StIdling           6
// StStopping         7
OUT:  A     #Ma.StStopped;
      L     1;	//Code=StStopped
      JC    Code;
      A     #Ma.StStarted;
      AN    #Ma.OutWarning;
      L     3;	//Code=StStarted
      JC    Code;
      A     #Ma.StStarted;
      A     #Ma.OutWarning;
      L     4;	//Code=StWarning 
      JC    Code;
      A     #Ma.StIdling;
      L     6;	//Code=StIdling
      JC    Code;
      A     #Ma.StStarting;
      L     2;	//Code=StStarting
      JC    Code;
      A     #Ma.StStopping;
      L     7;	//Code=StStopping 
      JC    Code;
      L     32;	//Code=StFault 
Code: L     #Ma.StCode;	// Old state code
      TAK;
      T     #Ma.StCode;	// Save state code
      <>I;
      L     3;
      CC    "SYS_CBitCtrl";	//Set change bit
NETWORK
TITLE = Global End
      CLR;	//---Clear all commands
      =     #Ma.CmdOnMan;
      =     #Ma.CmdOffMan;
      =     #Ma.CmdNext;
      =     #Ma.CmdFaultReset;
      =     #Ma.CmdFanOffMan;
END_FUNCTION_BLOCK

